C09088=1094.562,101.810,-61.706,176.099,17.273,152.460
C09089=1094.567,102.058,-61.724,176.101,17.273,152.459
C09090=1094.573,102.308,-61.742,176.104,17.274,152.459
C09091=1094.578,102.557,-61.761,176.106,17.275,152.459
C09092=1094.585,102.807,-61.779,176.108,17.276,152.458
C09093=1094.590,103.055,-61.798,176.111,17.277,152.458
C09094=1094.596,103.305,-61.816,176.113,17.277,152.458
C09095=1094.601,103.554,-61.835,176.116,17.279,152.457
C09096=1094.607,103.804,-61.853,176.119,17.279,152.457
C09097=1094.612,104.053,-61.871,176.121,17.280,152.457
C09098=1094.618,104.302,-61.890,176.123,17.281,152.457
C09099=1094.623,104.551,-61.909,176.126,17.281,152.456
C09100=1094.629,104.801,-61.926,176.128,17.283,152.456
C09101=1094.635,105.050,-61.946,176.131,17.284,152.456
C09102=1094.641,105.299,-61.963,176.133,17.284,152.455
C09103=1094.646,105.549,-61.983,176.136,17.285,152.455
C09104=1094.652,105.798,-62.000,176.138,17.286,152.455
C09105=1094.657,106.047,-62.019,176.141,17.287,152.454
C09106=1094.662,106.296,-62.037,176.144,17.288,152.454
C09107=1094.669,106.545,-62.056,176.145,17.288,152.454
C09108=1094.674,106.794,-62.075,176.148,17.289,152.453
C09109=1094.680,107.044,-62.093,176.151,17.290,152.453
C09110=1094.686,107.293,-62.112,176.153,17.291,152.453
C09111=1094.691,107.542,-62.130,176.156,17.292,152.452
C09112=1094.697,107.792,-62.149,176.158,17.292,152.452
C09113=1094.702,108.041,-62.168,176.161,17.293,152.452
C09114=1094.708,108.290,-62.186,176.164,17.294,152.451
C09115=1094.714,108.540,-62.205,176.166,17.295,152.451
C09116=1094.719,108.788,-62.223,176.169,17.296,152.451
C09117=1094.725,109.038,-62.243,176.171,17.296,152.450
C09118=1094.731,109.288,-62.261,176.173,17.297,152.450
C09119=1094.736,109.536,-62.279,176.176,17.298,152.450
C09120=1094.742,109.786,-62.299,176.178,17.299,152.449
C09121=1094.748,110.035,-62.317,176.181,17.300,152.449
C09122=1094.753,110.284,-62.335,176.184,17.301,152.449
C09123=1094.759,110.533,-62.355,176.186,17.301,152.449
C09124=1094.765,110.783,-62.373,176.189,17.302,152.448
C09125=1094.770,111.032,-62.391,176.191,17.302,152.448
C09126=1094.776,111.281,-62.411,176.194,17.303,152.447
C09127=1094.782,111.556,-62.431,176.197,17.304,152.447
C09128=1094.789,111.832,-62.452,176.199,17.305,152.447
C09129=1094.795,112.107,-62.473,176.202,17.306,152.446
C09130=1094.801,112.383,-62.494,176.205,17.307,152.446
C09131=1094.807,112.632,-62.512,176.207,17.307,152.446
C09132=1094.812,112.882,-62.531,176.210,17.308,152.445
C09133=1094.818,113.131,-62.550,176.213,17.309,152.445
C09134=1094.824,113.381,-62.570,176.215,17.310,152.445
C09135=1094.829,113.629,-62.588,176.218,17.311,152.444
C09136=1094.835,113.878,-62.607,176.220,17.311,152.444
C09137=1094.841,114.128,-62.626,176.223,17.312,152.443
C09138=1094.846,114.377,-62.645,176.226,17.313,152.443
C09139=1094.852,114.626,-62.664,176.228,17.313,152.443
C09140=1094.858,114.876,-62.682,176.231,17.314,152.443
C09141=1094.863,115.125,-62.701,176.234,17.315,152.442
C09142=1094.868,115.374,-62.720,176.236,17.316,152.442
C09143=1094.874,115.623,-62.740,176.239,17.316,152.441
C09144=1094.879,115.872,-62.759,176.241,17.318,152.441
C09145=1094.885,116.122,-62.778,176.243,17.318,152.441
C09146=1094.891,116.371,-62.797,176.246,17.319,152.441
C09147=1094.896,116.620,-62.816,176.249,17.320,152.440
C09148=1094.901,116.869,-62.835,176.251,17.321,152.440
C09149=1094.907,117.119,-62.854,176.254,17.321,152.439
C09150=1094.912,117.367,-62.873,176.257,17.322,152.439
C09151=1094.918,117.617,-62.893,176.259,17.323,152.439
C09152=1094.924,117.866,-62.912,176.262,17.323,152.438
C09153=1094.929,118.116,-62.931,176.265,17.325,152.438
C09154=1094.934,118.364,-62.950,176.267,17.325,152.438
C09155=1094.940,118.614,-62.969,176.270,17.326,152.437
C09156=1094.946,118.863,-62.988,176.273,17.327,152.437
C09157=1094.952,119.112,-63.007,176.275,17.327,152.437
C09158=1094.957,119.361,-63.026,176.278,17.328,152.436
C09159=1094.963,119.611,-63.045,176.280,17.328,152.436
C09160=1094.969,119.859,-63.065,176.283,17.329,152.436
C09161=1094.974,120.108,-63.084,176.286,17.330,152.435
C09162=1094.980,120.357,-63.103,176.287,17.331,152.435
C09163=1094.985,120.607,-63.122,176.290,17.331,152.434
C09164=1094.991,120.856,-63.142,176.293,17.332,152.434
C09165=1094.997,121.106,-63.161,176.295,17.333,152.434
C09166=1095.002,121.355,-63.180,176.298,17.333,152.433
C09167=1095.007,121.604,-63.200,176.301,17.334,152.433
C09168=1095.013,121.853,-63.220,176.303,17.335,152.433
C09169=1095.018,122.103,-63.239,176.306,17.336,152.432
C09170=1095.024,122.352,-63.258,176.309,17.336,152.432
C09171=1095.029,122.601,-63.277,176.311,17.337,152.432
C09172=1095.035,122.849,-63.297,176.314,17.338,152.431
C09173=1095.041,123.099,-63.316,176.317,17.338,152.431
C09174=1095.047,123.348,-63.335,176.319,17.339,152.430
C09175=1095.052,123.598,-63.355,176.322,17.339,152.430
C09176=1095.058,123.847,-63.375,176.325,17.340,152.430
C09177=1095.063,124.095,-63.394,176.327,17.341,152.429
C09178=1095.069,124.345,-63.413,176.330,17.342,152.429
C09179=1095.075,124.594,-63.432,176.333,17.342,152.429
C09180=1095.081,124.843,-63.452,176.336,17.343,152.428
C09181=1095.086,125.092,-63.471,176.338,17.343,152.428
C09182=1095.092,125.342,-63.490,176.341,17.345,152.427
C09183=1095.098,125.591,-63.510,176.344,17.345,152.427
C09184=1095.103,125.840,-63.530,176.346,17.345,152.427
C09185=1095.108,126.089,-63.549,176.349,17.346,152.426
C09186=1095.114,126.338,-63.569,176.352,17.347,152.426
C09187=1095.120,126.587,-63.588,176.354,17.347,152.425
C09188=1095.125,126.837,-63.608,176.357,17.348,152.425
C09189=1095.131,127.086,-63.628,176.360,17.349,152.425
C09190=1095.137,127.335,-63.647,176.362,17.349,152.424
C09191=1095.144,127.610,-63.669,176.365,17.350,152.424
C09192=1095.150,127.887,-63.691,176.368,17.350,152.423
C09193=1095.156,128.161,-63.712,176.371,17.351,152.423
C09194=1095.162,128.437,-63.733,176.374,17.352,152.422
C09195=1095.168,128.686,-63.753,176.377,17.353,152.422
C09196=1095.174,128.935,-63.772,176.380,17.353,152.422
C09197=1095.179,129.184,-63.793,176.383,17.354,152.421
C09198=1095.185,129.434,-63.812,176.386,17.354,152.421
C09199=1095.191,129.683,-63.832,176.389,17.355,152.420
C09200=1095.196,129.932,-63.851,176.391,17.355,152.420
C09201=1095.202,130.181,-63.871,176.394,17.356,152.420
C09202=1095.208,130.430,-63.891,176.397,17.357,152.419
C09203=1095.213,130.680,-63.911,176.399,17.357,152.419
C09204=1095.219,130.929,-63.930,176.402,17.358,152.418
C09205=1095.225,131.178,-63.950,176.405,17.358,152.418
C09206=1095.231,131.427,-63.970,176.407,17.359,152.418
C09207=1095.237,131.676,-63.990,176.410,17.359,152.417
C09208=1095.242,131.925,-64.010,176.413,17.360,152.417
C09209=1095.248,132.175,-64.029,176.416,17.361,152.416
C09210=1095.254,132.423,-64.049,176.418,17.361,152.416
C09211=1095.259,132.673,-64.070,176.421,17.362,152.415
C09212=1095.265,132.922,-64.089,176.424,17.363,152.415
C09213=1095.271,133.171,-64.109,176.426,17.363,152.415
C09214=1095.275,133.421,-64.129,176.429,17.364,152.414
C09215=1095.281,133.669,-64.149,176.432,17.364,152.414
C09216=1095.287,133.918,-64.169,176.434,17.364,152.413
C09217=1095.292,134.168,-64.189,176.437,17.365,152.413
C09218=1095.298,134.417,-64.209,176.440,17.366,152.413
C09219=1095.304,134.666,-64.229,176.443,17.367,152.412
C09220=1095.309,134.915,-64.248,176.446,17.367,152.412
C09221=1095.315,135.164,-64.268,176.449,17.367,152.411
C09222=1095.321,135.413,-64.289,176.452,17.368,152.411
C09223=1095.327,135.662,-64.309,176.454,17.368,152.410
C09224=1095.332,135.912,-64.329,176.457,17.369,152.410
C09225=1095.338,136.161,-64.349,176.460,17.370,152.410
C09226=1095.343,136.410,-64.369,176.463,17.370,152.409
C09227=1095.349,136.658,-64.389,176.465,17.371,152.409
C09228=1095.354,136.908,-64.409,176.468,17.371,152.408
C09229=1095.360,137.157,-64.429,176.471,17.372,152.408
C09230=1095.366,137.406,-64.449,176.473,17.372,152.408
C09231=1095.371,137.655,-64.470,176.476,17.373,152.407
C09232=1095.378,137.905,-64.490,176.479,17.373,152.407
C09233=1095.383,138.154,-64.510,176.482,17.374,152.406
C09234=1095.389,138.403,-64.530,176.485,17.374,152.406
C09235=1095.394,138.652,-64.550,176.488,17.375,152.405
C09236=1095.400,138.901,-64.570,176.491,17.376,152.405
C09237=1095.405,139.150,-64.591,176.494,17.376,152.404
C09238=1095.411,139.399,-64.611,176.496,17.376,152.404
C09239=1095.416,139.649,-64.631,176.499,17.377,152.404
C09240=1095.422,139.897,-64.651,176.502,17.378,152.403
C09241=1095.427,140.147,-64.671,176.504,17.378,152.403
C09242=1095.433,140.395,-64.691,176.507,17.378,152.402
C09243=1095.439,140.645,-64.712,176.510,17.379,152.402
C09244=1095.444,140.894,-64.733,176.513,17.380,152.401
C09245=1095.450,141.143,-64.752,176.516,17.380,152.401
C09246=1095.456,141.392,-64.773,176.519,17.381,152.401
C09247=1095.462,141.641,-64.793,176.522,17.382,152.400
C09248=1095.467,141.890,-64.814,176.525,17.382,152.400
C09249=1095.472,142.139,-64.834,176.527,17.382,152.399
C09250=1095.478,142.388,-64.854,176.530,17.383,152.399
C09251=1095.483,142.637,-64.875,176.533,17.384,152.398
C09252=1095.489,142.887,-64.896,176.536,17.384,152.398
C09253=1095.495,143.136,-64.915,176.538,17.384,152.397
C09254=1095.500,143.385,-64.936,176.541,17.385,152.397
C09255=1095.506,143.661,-64.959,176.545,17.385,152.396
C09256=1095.512,143.936,-64.981,176.548,17.386,152.396
C09257=1095.519,144.211,-65.004,176.551,17.386,152.395
C09258=1095.525,144.487,-65.026,176.554,17.387,152.395
C09259=1095.531,144.736,-65.047,176.557,17.388,152.395
C09260=1095.536,144.985,-65.067,176.560,17.388,152.394
C09261=1095.542,145.234,-65.088,176.562,17.388,152.394
C09262=1095.548,145.483,-65.108,176.565,17.389,152.393
C09263=1095.553,145.732,-65.129,176.569,17.389,152.393
C09264=1095.559,145.981,-65.149,176.572,17.390,152.392
C09265=1095.565,146.230,-65.170,176.574,17.390,152.392
C09266=1095.570,146.480,-65.191,176.577,17.391,152.391
C09267=1095.576,146.729,-65.211,176.580,17.391,152.391
C09268=1095.582,146.978,-65.231,176.583,17.392,152.390
C09269=1095.587,147.226,-65.253,176.585,17.392,152.390
C09270=1095.592,147.475,-65.273,176.588,17.393,152.390
C09271=1095.598,147.725,-65.294,176.592,17.393,152.389
C09272=1095.604,147.974,-65.314,176.595,17.394,152.389
C09273=1095.610,148.222,-65.335,176.597,17.393,152.388
C09274=1095.615,148.472,-65.356,176.600,17.394,152.388
C09275=1095.621,148.721,-65.377,176.603,17.395,152.387
C09276=1095.626,148.971,-65.397,176.606,17.395,152.387
C09277=1095.633,149.219,-65.418,176.608,17.395,152.386
C09278=1095.638,149.468,-65.439,176.612,17.396,152.386
C09279=1095.644,149.718,-65.460,176.615,17.397,152.385
C09280=1095.649,149.967,-65.480,176.618,17.397,152.385
C09281=1095.654,150.215,-65.501,176.621,17.398,152.384
C09282=1095.660,150.464,-65.522,176.623,17.398,152.384
C09283=1095.666,150.714,-65.543,176.626,17.398,152.383
C09284=1095.671,150.963,-65.564,176.629,17.399,152.383
C09285=1095.677,151.212,-65.584,176.632,17.400,152.382
C09286=1095.682,151.461,-65.605,176.635,17.399,152.382
C09287=1095.689,151.710,-65.626,176.638,17.400,152.382
C09288=1095.694,151.959,-65.647,176.641,17.400,152.381
C09289=1095.699,152.208,-65.668,176.644,17.401,152.381
C09290=1095.705,152.457,-65.689,176.647,17.402,152.380
C09291=1095.711,152.706,-65.710,176.649,17.402,152.380
C09292=1095.716,152.955,-65.731,176.653,17.402,152.379
C09293=1095.722,153.205,-65.752,176.656,17.403,152.379
C09294=1095.727,153.453,-65.773,176.659,17.403,152.378
C09295=1095.733,153.702,-65.794,176.661,17.403,152.378
C09296=1095.739,153.952,-65.815,176.664,17.404,152.377
C09297=1095.744,154.201,-65.836,176.667,17.404,152.377
C09298=1095.750,154.449,-65.857,176.671,17.405,152.376
C09299=1095.756,154.699,-65.878,176.674,17.405,152.376
C09300=1095.761,154.948,-65.899,176.676,17.405,152.375
C09301=1095.766,155.197,-65.920,176.679,17.405,152.375
C09302=1095.773,155.446,-65.941,176.682,17.406,152.374
C09303=1095.778,155.695,-65.962,176.686,17.407,152.374
C09304=1095.783,155.944,-65.983,176.688,17.407,152.373
C09305=1095.789,156.193,-66.004,176.691,17.407,152.373
C09306=1095.795,156.442,-66.025,176.694,17.408,152.372
C09307=1095.800,156.690,-66.047,176.697,17.408,152.372
C09308=1095.806,156.940,-66.068,176.700,17.409,152.371
C09309=1095.812,157.189,-66.089,176.703,17.409,152.371
C09310=1095.817,157.438,-66.109,176.706,17.409,152.370
C09311=1095.823,157.687,-66.131,176.709,17.410,152.370
C09312=1095.828,157.936,-66.153,176.712,17.410,152.369
C09313=1095.834,158.186,-66.174,176.715,17.411,152.369
C09314=1095.839,158.434,-66.195,176.718,17.411,152.368
C09315=1095.845,158.683,-66.216,176.721,17.411,152.368
C09316=1095.851,158.933,-66.237,176.724,17.412,152.367
C09317=1095.856,159.181,-66.259,176.727,17.412,152.367
C09318=1095.863,159.430,-66.280,176.730,17.412,152.366
C09319=1095.868,159.706,-66.304,176.734,17.413,152.366
C09320=1095.874,159.981,-66.327,176.737,17.413,152.365
C09321=1095.881,160.255,-66.350,176.740,17.413,152.364
C09322=1095.888,160.531,-66.374,176.743,17.414,152.364
C09323=1095.892,160.780,-66.396,176.746,17.414,152.363
C09324=1095.898,161.029,-66.417,176.750,17.415,152.363
C09325=1095.904,161.278,-66.438,176.752,17.414,152.362
C09326=1095.909,161.527,-66.459,176.755,17.415,152.362
C09327=1095.916,161.776,-66.481,176.758,17.415,152.361
C09328=1095.920,162.025,-66.503,176.761,17.416,152.361
C09329=1095.927,162.274,-66.525,176.764,17.417,152.360
C09330=1095.931,162.524,-66.546,176.768,17.417,152.360
C09331=1095.937,162.772,-66.567,176.770,17.417,152.359
C09332=1095.943,163.021,-66.589,176.773,17.417,152.359
C09333=1095.948,163.270,-66.610,176.776,17.418,152.358
C09334=1095.954,163.519,-66.632,176.779,17.419,152.358
C09335=1095.959,163.768,-66.654,176.783,17.419,152.357
C09336=1095.964,164.017,-66.675,176.786,17.419,152.357
C09337=1095.970,164.266,-66.696,176.788,17.419,152.356
C09338=1095.975,164.515,-66.718,176.791,17.420,152.356
C09339=1095.981,164.764,-66.740,176.795,17.420,152.355
C09340=1095.986,165.013,-66.762,176.798,17.421,152.355
C09341=1095.992,165.262,-66.783,176.801,17.421,152.354
C09342=1095.997,165.511,-66.805,176.804,17.421,152.354
C09343=1096.003,165.760,-66.827,176.806,17.422,152.353
C09344=1096.008,166.009,-66.848,176.809,17.422,152.353
C09345=1096.013,166.258,-66.870,176.813,17.422,152.352
C09346=1096.019,166.507,-66.891,176.816,17.423,152.352
C09347=1096.024,166.756,-66.913,176.819,17.423,152.351
C09348=1096.030,167.005,-66.935,176.822,17.424,152.351
C09349=1096.035,167.254,-66.957,176.825,17.423,152.350
C09350=1096.041,167.503,-66.978,176.828,17.424,152.350
C09351=1096.046,167.752,-67.000,176.831,17.425,152.349
C09352=1096.052,168.001,-67.022,176.834,17.425,152.349
C09353=1096.058,168.251,-67.044,176.837,17.425,152.348
C09354=1096.063,168.499,-67.065,176.841,17.425,152.348
C09355=1096.069,168.749,-67.088,176.843,17.425,152.347
C09356=1096.074,168.997,-67.109,176.846,17.426,152.347
C09357=1096.080,169.247,-67.131,176.849,17.426,152.346
C09358=1096.086,169.494,-67.153,176.853,17.427,152.345
C09359=1096.091,169.744,-67.175,176.856,17.427,152.345
C09360=1096.097,169.992,-67.197,176.859,17.427,152.344
C09361=1096.102,170.242,-67.219,176.862,17.428,152.344
C09362=1096.108,170.491,-67.240,176.865,17.428,152.343
C09363=1096.113,170.740,-67.262,176.868,17.428,152.343
C09364=1096.119,170.989,-67.284,176.871,17.428,152.342
C09365=1096.124,171.237,-67.307,176.874,17.429,152.342
C09366=1096.130,171.487,-67.329,176.878,17.429,152.341
C09367=1096.135,171.735,-67.350,176.881,17.429,152.341
C09368=1096.141,171.985,-67.372,176.884,17.430,152.340
C09369=1096.147,172.234,-67.395,176.887,17.430,152.340
C09370=1096.152,172.482,-67.417,176.890,17.430,152.339
C09371=1096.158,172.732,-67.438,176.893,17.430,152.338
C09372=1096.164,172.981,-67.460,176.896,17.431,152.338
C09373=1096.169,173.229,-67.483,176.900,17.431,152.337
C09374=1096.175,173.478,-67.505,176.903,17.432,152.337
C09375=1096.180,173.728,-67.527,176.906,17.432,152.336
C09376=1096.186,173.976,-67.549,176.908,17.432,152.336
C09377=1096.192,174.225,-67.571,176.911,17.432,152.335
C09378=1096.197,174.475,-67.593,176.915,17.432,152.335
C09379=1096.203,174.723,-67.615,176.918,17.433,152.334
C09380=1096.208,174.972,-67.637,176.921,17.433,152.334
C09381=1096.215,175.222,-67.659,176.924,17.433,152.333
C09382=1096.220,175.470,-67.682,176.928,17.434,152.332
C09383=1096.226,175.745,-67.707,176.931,17.434,152.332
C09384=1096.232,176.020,-67.731,176.935,17.434,152.331
C09385=1096.239,176.294,-67.755,176.938,17.434,152.330
C09386=1096.245,176.570,-67.780,176.941,17.434,152.330
C09387=1096.250,176.818,-67.802,176.945,17.434,152.329
C09388=1096.256,177.067,-67.824,176.948,17.435,152.329
C09389=1096.262,177.316,-67.846,176.951,17.435,152.328
C09390=1096.267,177.565,-67.869,176.954,17.435,152.328
C09391=1096.273,177.814,-67.891,176.958,17.436,152.327
C09392=1096.279,178.063,-67.914,176.961,17.436,152.327
C09393=1096.284,178.312,-67.936,176.964,17.435,152.326
C09394=1096.291,178.561,-67.958,176.967,17.436,152.325
C09395=1096.295,178.810,-67.980,176.970,17.436,152.325
C09396=1096.301,179.059,-68.003,176.973,17.436,152.324
C09397=1096.307,179.308,-68.025,176.977,17.437,152.324
C09398=1096.313,179.557,-68.048,176.980,17.437,152.323
C09399=1096.318,179.805,-68.069,176.983,17.437,152.322
C09400=1096.324,180.054,-68.092,176.987,17.437,152.322
C09401=1096.330,180.303,-68.115,176.989,17.437,152.321
C09402=1096.336,180.552,-68.137,176.992,17.437,152.321
C09403=1096.341,180.801,-68.160,176.996,17.438,152.320
C09404=1096.347,181.050,-68.183,176.999,17.438,152.320
C09405=1096.353,181.299,-68.204,177.002,17.438,152.319
C09406=1096.358,181.548,-68.227,177.006,17.438,152.318
C09407=1096.364,181.797,-68.250,177.009,17.439,152.318
C09408=1096.369,182.046,-68.272,177.012,17.439,152.317
C09409=1096.376,182.295,-68.295,177.015,17.439,152.317
C09410=1096.382,182.544,-68.318,177.018,17.439,152.316
C09411=1096.387,182.793,-68.340,177.021,17.439,152.315
C09412=1096.392,183.041,-68.362,177.025,17.439,152.315
C09413=1096.399,183.290,-68.385,177.028,17.440,152.314
C09414=1096.404,183.539,-68.408,177.031,17.439,152.314
C09415=1096.410,183.788,-68.430,177.035,17.440,152.313
C09416=1096.416,184.037,-68.453,177.038,17.440,152.312
C09417=1096.421,184.286,-68.476,177.041,17.440,152.312
C09418=1096.428,184.535,-68.498,177.045,17.440,152.311
C09419=1096.433,184.784,-68.520,177.048,17.441,152.311
C09420=1096.439,185.033,-68.543,177.051,17.440,152.310
C09421=1096.445,185.282,-68.566,177.054,17.440,152.309
C09422=1096.450,185.530,-68.589,177.057,17.441,152.309
C09423=1096.456,185.779,-68.612,177.060,17.441,152.308
C09424=1096.461,186.028,-68.635,177.064,17.441,152.308
C09425=1096.467,186.277,-68.657,177.067,17.442,152.307
C09426=1096.472,186.527,-68.680,177.070,17.442,152.307
C09427=1096.477,186.775,-68.703,177.074,17.442,152.306
C09428=1096.483,187.024,-68.726,177.077,17.442,152.305
C09429=1096.488,187.273,-68.749,177.080,17.443,152.305
C09430=1096.494,187.522,-68.772,177.083,17.443,152.304
C09431=1096.500,187.770,-68.795,177.087,17.443,152.304
C09432=1096.505,188.019,-68.818,177.090,17.444,152.303
C09433=1096.511,188.268,-68.841,177.093,17.444,152.302
C09434=1096.516,188.517,-68.864,177.096,17.443,152.302
C09435=1096.521,188.766,-68.886,177.099,17.444,152.301
C09436=1096.527,189.015,-68.909,177.102,17.444,152.301
C09437=1096.532,189.264,-68.932,177.106,17.444,152.300
C09438=1096.538,189.513,-68.955,177.109,17.444,152.300
C09439=1096.544,189.762,-68.978,177.112,17.445,152.299
C09440=1096.549,190.011,-69.001,177.116,17.445,152.298
C09441=1096.555,190.259,-69.025,177.119,17.445,152.298
C09442=1096.561,190.508,-69.048,177.122,17.445,152.297
C09443=1096.566,190.756,-69.071,177.126,17.445,152.297
C09444=1096.572,191.005,-69.094,177.129,17.446,152.296
C09445=1096.577,191.255,-69.117,177.132,17.446,152.295
C09446=1096.582,191.503,-69.140,177.136,17.446,152.295
C09447=1096.589,191.778,-69.166,177.139,17.446,152.294
C09448=1096.595,192.052,-69.191,177.142,17.446,152.293
C09449=1096.601,192.327,-69.217,177.146,17.446,152.293
C09450=1096.607,192.601,-69.242,177.150,17.447,152.292
C09451=1096.613,192.850,-69.265,177.154,17.447,152.291
C09452=1096.619,193.099,-69.288,177.157,17.447,152.291
C09453=1096.624,193.348,-69.312,177.160,17.447,152.290
C09454=1096.630,193.597,-69.335,177.164,17.448,152.290
C09455=1096.635,193.846,-69.358,177.166,17.447,152.289
C09456=1096.641,194.094,-69.381,177.170,17.447,152.288
C09457=1096.646,194.344,-69.405,177.173,17.448,152.288
C09458=1096.652,194.593,-69.428,177.176,17.448,152.287
C09459=1096.658,194.841,-69.451,177.180,17.448,152.287
C09460=1096.664,195.090,-69.475,177.183,17.448,152.286
C09461=1096.669,195.339,-69.498,177.186,17.448,152.285
C09462=1096.675,195.588,-69.521,177.190,17.448,152.285
C09463=1096.680,195.837,-69.544,177.193,17.449,152.284
C09464=1096.686,196.085,-69.568,177.196,17.449,152.284
C09465=1096.691,196.334,-69.591,177.200,17.449,152.283
C09466=1096.697,196.583,-69.614,177.203,17.449,152.282
C09467=1096.702,196.832,-69.638,177.206,17.449,152.282
C09468=1096.708,197.081,-69.661,177.210,17.449,152.281
C09469=1096.714,197.329,-69.684,177.213,17.450,152.280
C09470=1096.719,197.578,-69.708,177.216,17.450,152.280
C09471=1096.725,197.828,-69.732,177.220,17.450,152.279
C09472=1096.731,198.076,-69.755,177.223,17.450,152.279
C09473=1096.736,198.325,-69.779,177.227,17.450,152.278
C09474=1096.742,198.574,-69.802,177.230,17.450,152.277
C09475=1096.748,198.822,-69.826,177.233,17.450,152.277
C09476=1096.753,199.072,-69.849,177.237,17.451,152.276
C09477=1096.759,199.320,-69.873,177.240,17.451,152.275
C09478=1096.765,199.569,-69.896,177.243,17.451,152.275
C09479=1096.771,199.818,-69.920,177.247,17.451,152.274
C09480=1096.777,200.067,-69.943,177.250,17.451,152.274
C09481=1096.783,200.315,-69.967,177.254,17.451,152.273
C09482=1096.788,200.564,-69.991,177.257,17.451,152.272
C09483=1096.794,200.813,-70.014,177.261,17.451,152.272
C09484=1096.799,201.062,-70.038,177.264,17.451,152.271
C09485=1096.805,201.311,-70.062,177.267,17.452,152.270
C09486=1096.811,201.560,-70.085,177.271,17.452,152.270
C09487=1096.816,201.808,-70.109,177.274,17.452,152.269
C09488=1096.822,202.057,-70.133,177.277,17.451,152.269
C09489=1096.827,202.306,-70.156,177.280,17.451,152.268
C09490=1096.834,202.555,-70.180,177.284,17.452,152.267
C09491=1096.839,202.804,-70.204,177.287,17.451,152.267
C09492=1096.845,203.052,-70.227,177.290,17.452,152.266
C09493=1096.850,203.301,-70.252,177.294,17.452,152.265
C09494=1096.856,203.550,-70.275,177.297,17.452,152.265
C09495=1096.861,203.798,-70.299,177.301,17.452,152.264
C09496=1096.867,204.048,-70.323,177.304,17.452,152.263
C09497=1096.873,204.297,-70.346,177.307,17.452,152.263
C09498=1096.878,204.545,-70.371,177.311,17.453,152.262
C09499=1096.884,204.793,-70.394,177.314,17.453,152.262
C09500=1096.889,205.043,-70.418,177.318,17.454,152.261
C09501=1096.895,205.292,-70.442,177.322,17.453,152.260
C09502=1096.901,205.540,-70.466,177.325,17.453,152.260
C09503=1096.906,205.789,-70.490,177.328,17.454,152.259
C09504=1096.912,206.038,-70.514,177.332,17.454,152.258
C09505=1096.918,206.286,-70.538,177.335,17.454,152.258
C09506=1096.923,206.535,-70.562,177.339,17.454,152.257
C09507=1096.929,206.784,-70.586,177.342,17.454,152.257
C09508=1096.935,207.033,-70.609,177.346,17.454,152.256
C09509=1096.940,207.282,-70.634,177.349,17.454,152.255
C09510=1096.946,207.531,-70.658,177.352,17.454,152.255
C09511=1096.969,208.543,-70.756,177.400,17.473,152.249
C09512=1096.977,208.915,-70.792,177.405,17.474,152.249
C09513=1096.986,209.287,-70.828,177.410,17.476,152.248
C09514=1096.994,209.658,-70.865,177.415,17.477,152.247
C09515=1097.002,210.030,-70.901,177.420,17.479,152.247
C09516=1097.008,210.280,-70.926,177.423,17.479,152.246
C09517=1097.013,210.528,-70.950,177.426,17.480,152.246
C09518=1097.019,210.777,-70.975,177.430,17.482,152.246
C09519=1097.025,211.026,-70.999,177.433,17.482,152.245
C09520=1097.030,211.275,-71.023,177.436,17.483,152.245
C09521=1097.036,211.524,-71.048,177.439,17.485,152.244
C09522=1097.041,211.772,-71.073,177.442,17.486,152.244
C09523=1097.047,212.020,-71.097,177.445,17.486,152.244
C09524=1097.053,212.270,-71.122,177.449,17.488,152.243
C09525=1097.058,212.518,-71.146,177.452,17.489,152.243
C09526=1097.065,212.767,-71.170,177.455,17.489,152.242
C09527=1097.070,213.015,-71.195,177.459,17.491,152.242
C09528=1097.076,213.265,-71.220,177.462,17.491,152.241
C09529=1097.081,213.513,-71.244,177.465,17.492,152.241
C09530=1097.086,213.762,-71.269,177.469,17.494,152.241
C09531=1097.092,214.011,-71.294,177.472,17.494,152.240
C09532=1097.097,214.259,-71.319,177.475,17.495,152.240
C09533=1097.103,214.509,-71.343,177.478,17.497,152.239
C09534=1097.109,214.757,-71.368,177.481,17.497,152.239
C09535=1097.114,215.005,-71.392,177.484,17.498,152.239
C09536=1097.120,215.254,-71.417,177.488,17.500,152.238
C09537=1097.126,215.502,-71.442,177.491,17.501,152.238
C09538=1097.132,215.752,-71.467,177.494,17.501,152.237
C09539=1097.136,216.001,-71.491,177.498,17.503,152.237
C09540=1097.142,216.249,-71.517,177.501,17.504,152.237
C09541=1097.148,216.498,-71.541,177.504,17.505,152.236
C09542=1097.154,216.747,-71.566,177.507,17.506,152.236
C09543=1097.159,216.995,-71.591,177.510,17.507,152.235
C09544=1097.165,217.244,-71.615,177.514,17.508,152.235
C09545=1097.171,217.492,-71.640,177.517,17.509,152.235
C09546=1097.176,217.742,-71.665,177.520,17.510,152.234
C09547=1097.182,217.990,-71.690,177.524,17.511,152.234
C09548=1097.187,218.239,-71.715,177.527,17.512,152.233
C09549=1097.193,218.487,-71.740,177.530,17.513,152.233
C09550=1097.199,218.737,-71.765,177.534,17.514,152.232
C09551=1097.204,218.985,-71.790,177.537,17.515,152.232
C09552=1097.210,219.234,-71.815,177.541,17.516,152.232
C09553=1097.215,219.482,-71.840,177.544,17.517,152.231
C09554=1097.221,219.731,-71.864,177.546,17.518,152.231
C09555=1097.227,219.980,-71.890,177.550,17.519,152.230
C09556=1097.232,220.229,-71.915,177.553,17.520,152.230
C09557=1097.238,220.478,-71.940,177.556,17.521,152.230
C09558=1097.244,220.726,-71.965,177.560,17.522,152.229
C09559=1097.250,220.975,-71.990,177.563,17.523,152.229
C09560=1097.255,221.223,-72.015,177.567,17.525,152.228
C09561=1097.260,221.472,-72.040,177.570,17.525,152.228
C09562=1097.267,221.721,-72.065,177.573,17.526,152.228
C09563=1097.272,221.969,-72.090,177.577,17.527,152.227
C09564=1097.281,222.345,-72.128,177.581,17.529,152.227
C09565=1097.288,222.721,-72.167,177.586,17.531,152.226
C09566=1097.297,223.097,-72.205,177.591,17.532,152.225
C09567=1097.305,223.473,-72.243,177.596,17.534,152.225
C09568=1097.312,223.721,-72.268,177.600,17.535,152.224
C09569=1097.317,223.971,-72.293,177.603,17.536,152.224
C09570=1097.322,224.219,-72.318,177.606,17.537,152.224
C09571=1097.329,224.467,-72.344,177.609,17.538,152.223
C09572=1097.333,224.716,-72.369,177.612,17.539,152.223
C09573=1097.339,224.965,-72.394,177.616,17.540,152.222
C09574=1097.345,225.214,-72.420,177.619,17.541,152.222
C09575=1097.350,225.462,-72.445,177.622,17.542,152.222
C09576=1097.356,225.711,-72.471,177.626,17.544,152.221
C09577=1097.362,225.960,-72.496,177.629,17.544,152.221
C09578=1097.367,226.208,-72.521,177.633,17.546,152.220
C09579=1097.373,226.457,-72.547,177.636,17.547,152.220
C09580=1097.379,226.706,-72.573,177.639,17.548,152.220
C09581=1097.384,226.954,-72.597,177.642,17.549,152.219
C09582=1097.389,227.203,-72.623,177.645,17.550,152.219
C09583=1097.396,227.452,-72.648,177.649,17.551,152.218
C09584=1097.401,227.701,-72.674,177.652,17.552,152.218
C09585=1097.407,227.949,-72.699,177.656,17.554,152.218
C09586=1097.412,228.198,-72.725,177.659,17.554,152.217
C09587=1097.418,228.446,-72.750,177.662,17.555,152.217
C09588=1097.423,228.695,-72.776,177.665,17.557,152.216
C09589=1097.429,228.943,-72.801,177.668,17.558,152.216
C09590=1097.435,229.192,-72.827,177.672,17.559,152.216
C09591=1097.441,229.441,-72.853,177.675,17.560,152.215
C09592=1097.446,229.689,-72.878,177.679,17.561,152.215
C09593=1097.452,229.938,-72.904,177.682,17.562,152.214
C09594=1097.458,230.187,-72.929,177.685,17.563,152.214
C09595=1097.463,230.435,-72.956,177.689,17.564,152.214
C09596=1097.470,230.684,-72.981,177.692,17.565,152.213
C09597=1097.475,230.932,-73.007,177.695,17.567,152.213
C09598=1097.480,231.181,-73.033,177.698,17.568,152.213
C09599=1097.486,231.430,-73.058,177.702,17.569,152.212
C09600=1097.492,231.679,-73.084,177.705,17.570,152.212
C09601=1097.497,231.927,-73.110,177.709,17.571,152.211
C09602=1097.503,232.176,-73.135,177.712,17.572,152.211
C09603=1097.509,232.424,-73.162,177.715,17.574,152.211
C09604=1097.514,232.673,-73.188,177.718,17.574,152.210
C09605=1097.519,232.922,-73.214,177.721,17.575,152.210
C09606=1097.525,233.170,-73.239,177.725,17.577,152.209
C09607=1097.531,233.418,-73.265,177.728,17.578,152.209
C09608=1097.536,233.667,-73.291,177.732,17.579,152.209
C09609=1097.542,233.916,-73.317,177.735,17.580,152.208
C09610=1097.548,234.165,-73.342,177.739,17.581,152.208
C09611=1097.553,234.413,-73.369,177.742,17.582,152.207
C09612=1097.559,234.662,-73.395,177.745,17.584,152.207
C09613=1097.564,234.911,-73.421,177.748,17.585,152.207
C09614=1097.570,235.159,-73.447,177.752,17.586,152.206
C09615=1097.576,235.408,-73.473,177.755,17.587,152.206
C09616=1097.584,235.775,-73.511,177.760,17.589,152.205
C09617=1097.592,236.143,-73.550,177.764,17.590,152.205
C09618=1097.600,236.509,-73.588,177.770,17.593,152.204
C09619=1097.608,236.878,-73.627,177.775,17.594,152.204
C09620=1097.615,237.126,-73.653,177.778,17.596,152.203
C09621=1097.620,237.374,-73.678,177.781,17.597,152.203
C09622=1097.625,237.622,-73.705,177.784,17.598,152.203
C09623=1097.631,237.871,-73.731,177.788,17.599,152.202
C09624=1097.637,238.120,-73.758,177.791,17.600,152.202
C09625=1097.642,238.369,-73.784,177.795,17.602,152.201
C09626=1097.648,238.617,-73.810,177.798,17.602,152.201
C09627=1097.653,238.866,-73.836,177.801,17.604,152.201
C09628=1097.659,239.114,-73.863,177.804,17.605,152.200
C09629=1097.665,239.363,-73.889,177.808,17.606,152.200
C09630=1097.670,239.612,-73.915,177.811,17.607,152.200
C09631=1097.677,239.860,-73.941,177.815,17.608,152.199
C09632=1097.682,240.109,-73.967,177.818,17.609,152.199
C09633=1097.688,240.357,-73.994,177.821,17.611,152.199
C09634=1097.693,240.605,-74.020,177.824,17.612,152.198
C09635=1097.699,240.854,-74.046,177.828,17.614,152.198
C09636=1097.704,241.103,-74.072,177.831,17.614,152.197
C09637=1097.710,241.351,-74.099,177.835,17.616,152.197
C09638=1097.716,241.599,-74.126,177.838,17.617,152.197
C09639=1097.721,241.848,-74.151,177.841,17.618,152.196
C09640=1097.727,242.097,-74.178,177.844,17.619,152.196
C09641=1097.733,242.345,-74.205,177.848,17.620,152.195
C09642=1097.739,242.593,-74.231,177.851,17.621,152.195
C09643=1097.743,242.843,-74.258,177.855,17.623,152.195
C09644=1097.749,243.091,-74.285,177.858,17.624,152.194
C09645=1097.755,243.339,-74.311,177.861,17.626,152.194
C09646=1097.761,243.588,-74.338,177.864,17.626,152.194
C09647=1097.766,243.837,-74.364,177.868,17.628,152.193
C09648=1097.772,244.085,-74.390,177.871,17.629,152.193
C09649=1097.778,244.333,-74.417,177.875,17.630,152.192
C09650=1097.783,244.582,-74.444,177.877,17.632,152.192
C09651=1097.788,244.830,-74.471,177.881,17.633,152.192
C09652=1097.794,245.079,-74.497,177.885,17.634,152.191
C09653=1097.800,245.328,-74.524,177.888,17.635,152.191
C09654=1097.805,245.576,-74.550,177.892,17.637,152.191
C09655=1097.811,245.825,-74.577,177.895,17.638,152.190
C09656=1097.817,246.074,-74.604,177.898,17.640,152.190
C09657=1097.823,246.322,-74.631,177.901,17.640,152.190
C09658=1097.828,246.571,-74.658,177.905,17.642,152.189
C09659=1097.834,246.819,-74.684,177.908,17.643,152.189
C09660=1097.839,247.068,-74.712,177.912,17.644,152.188
C09661=1097.845,247.317,-74.738,177.914,17.645,152.188
C09662=1097.851,247.565,-74.764,177.918,17.647,152.188
C09663=1097.856,247.814,-74.792,177.922,17.648,152.187
C09664=1097.861,248.062,-74.818,177.925,17.649,152.187
C09665=1097.867,248.310,-74.845,177.928,17.651,152.187
C09666=1097.872,248.559,-74.872,177.931,17.652,152.186
C09667=1097.878,248.807,-74.899,177.935,17.653,152.186
C09668=1097.886,249.168,-74.938,177.939,17.656,152.186
C09669=1097.895,249.528,-74.977,177.944,17.657,152.185
C09670=1097.902,249.889,-75.016,177.949,17.659,152.185
C09671=1097.910,250.249,-75.056,177.955,17.661,152.184
C09672=1097.916,250.497,-75.083,177.957,17.662,152.184
C09673=1097.921,250.746,-75.110,177.961,17.664,152.183
C09674=1097.927,250.994,-75.137,177.964,17.665,152.183
C09675=1097.932,251.243,-75.163,177.968,17.666,152.183
C09676=1097.937,251.491,-75.191,177.970,17.668,152.182
C09677=1097.944,251.740,-75.218,177.974,17.669,152.182
C09678=1097.949,251.988,-75.246,177.978,17.671,152.182
C09679=1097.955,252.237,-75.272,177.981,17.672,152.181
C09680=1097.960,252.485,-75.299,177.984,17.673,152.181
C09681=1097.966,252.734,-75.326,177.987,17.674,152.181
C09682=1097.971,252.982,-75.354,177.991,17.676,152.180
C09683=1097.977,253.231,-75.381,177.994,17.678,152.180
C09684=1097.983,253.480,-75.408,177.997,17.679,152.180
C09685=1097.989,253.727,-75.436,178.001,17.680,152.179
C09686=1097.994,253.976,-75.463,178.004,17.681,152.179
C09687=1097.999,254.224,-75.490,178.008,17.683,152.179
C09688=1098.005,254.473,-75.518,178.011,17.684,152.178
C09689=1098.011,254.721,-75.545,178.014,17.685,152.178
C09690=1098.016,254.970,-75.572,178.018,17.687,152.178
C09691=1098.022,255.218,-75.599,178.021,17.688,152.177
C09692=1098.027,255.467,-75.626,178.025,17.689,152.177
C09693=1098.034,255.716,-75.653,178.028,17.691,152.177
C09694=1098.039,255.964,-75.681,178.031,17.692,152.176
C09695=1098.044,256.212,-75.709,178.035,17.694,152.176
C09696=1098.050,256.460,-75.736,178.038,17.694,152.176
C09697=1098.056,256.709,-75.764,178.041,17.696,152.175
C09698=1098.062,256.957,-75.791,178.045,17.698,152.175
C09699=1098.067,257.206,-75.818,178.048,17.699,152.175
C09700=1098.074,257.454,-75.846,178.052,17.700,152.174
C09701=1098.079,257.703,-75.873,178.054,17.702,152.174
C09702=1098.084,257.951,-75.901,178.058,17.703,152.174
C09703=1098.090,258.199,-75.928,178.062,17.704,152.173
C09704=1098.096,258.448,-75.956,178.064,17.706,152.173
C09705=1098.101,258.696,-75.983,178.068,17.707,152.173
C09706=1098.107,258.945,-76.011,178.072,17.709,152.172
C09707=1098.113,259.193,-76.039,178.075,17.710,152.172
C09708=1098.118,259.442,-76.066,178.078,17.711,152.172
C09709=1098.124,259.690,-76.094,178.081,17.712,152.171
C09710=1098.129,259.939,-76.121,178.085,17.714,152.171
C09711=1098.136,260.187,-76.149,178.089,17.716,152.171
C09712=1098.141,260.436,-76.177,178.092,17.717,152.170
C09713=1098.147,260.684,-76.204,178.095,17.718,152.170
C09714=1098.153,260.932,-76.231,178.099,17.720,152.169
C09715=1098.159,261.181,-76.260,178.102,17.721,152.169
C09716=1098.164,261.429,-76.287,178.106,17.722,152.169
C09717=1098.170,261.677,-76.314,178.108,17.723,152.168
C09718=1098.176,261.926,-76.343,178.112,17.725,152.168
C09719=1098.181,262.174,-76.371,178.116,17.727,152.168
C09720=1098.190,262.531,-76.410,178.121,17.728,152.167
C09721=1098.197,262.889,-76.450,178.125,17.730,152.167
C09722=1098.207,263.247,-76.490,178.130,17.732,152.166
C09723=1098.215,263.605,-76.531,178.135,17.735,152.166
C09724=1098.220,263.853,-76.559,178.138,17.735,152.165
C09725=1098.227,264.101,-76.586,178.142,17.737,152.165
C09726=1098.232,264.349,-76.614,178.145,17.739,152.165
C09727=1098.238,264.598,-76.643,178.148,17.740,152.165
C09728=1098.243,264.847,-76.670,178.152,17.742,152.164
C09729=1098.248,265.095,-76.698,178.156,17.743,152.164
C09730=1098.254,265.343,-76.726,178.158,17.744,152.164
C09731=1098.259,265.591,-76.754,178.162,17.746,152.163
C09732=1098.265,265.840,-76.782,178.166,17.748,152.163
C09733=1098.271,266.088,-76.810,178.169,17.749,152.163
C09734=1098.276,266.336,-76.838,178.172,17.751,152.162
C09735=1098.282,266.585,-76.867,178.176,17.752,152.162
C09736=1098.287,266.833,-76.895,178.178,17.753,152.162
C09737=1098.293,267.082,-76.923,178.182,17.755,152.161
C09738=1098.299,267.330,-76.951,178.186,17.757,152.161
C09739=1098.305,267.579,-76.979,178.189,17.758,152.161
C09740=1098.310,267.827,-77.007,178.192,17.760,152.161
C09741=1098.316,268.075,-77.035,178.196,17.761,152.160
C09742=1098.321,268.323,-77.063,178.200,17.763,152.160
C09743=1098.328,268.572,-77.092,178.202,17.764,152.160
C09744=1098.333,268.820,-77.120,178.206,17.765,152.159
C09745=1098.339,269.068,-77.149,178.209,17.767,152.159
C09746=1098.344,269.316,-77.177,178.212,17.768,152.159
C09747=1098.350,269.565,-77.205,178.216,17.770,152.158
C09748=1098.355,269.813,-77.233,178.220,17.772,152.158
C09749=1098.361,270.062,-77.261,178.222,17.773,152.158
C09750=1098.367,270.309,-77.290,178.226,17.774,152.157
C09751=1098.373,270.558,-77.318,178.230,17.776,152.157
C09752=1098.378,270.806,-77.346,178.232,17.778,152.157
C09753=1098.384,271.055,-77.375,178.236,17.779,152.157
C09754=1098.390,271.302,-77.403,178.239,17.781,152.156
C09755=1098.395,271.551,-77.432,178.243,17.782,152.156
C09756=1098.400,271.800,-77.460,178.246,17.784,152.156
C09757=1098.406,272.048,-77.488,178.250,17.785,152.155
C09758=1098.413,272.296,-77.518,178.253,17.787,152.155
C09759=1098.418,272.544,-77.545,178.256,17.788,152.155
C09760=1098.424,272.793,-77.574,178.260,17.790,152.155
C09761=1098.429,273.041,-77.603,178.263,17.792,152.154
C09762=1098.435,273.290,-77.631,178.267,17.793,152.154
C09763=1098.440,273.538,-77.659,178.269,17.795,152.154
C09764=1098.446,273.786,-77.688,178.273,17.796,152.153
C09765=1098.452,274.035,-77.717,178.277,17.798,152.153
C09766=1098.457,274.282,-77.746,178.280,17.800,152.153
C09767=1098.463,274.531,-77.774,178.283,17.801,152.153
C09768=1098.468,274.779,-77.802,178.287,17.803,152.152
C09769=1098.475,275.027,-77.831,178.290,17.805,152.152
C09770=1098.480,275.276,-77.860,178.293,17.806,152.152
C09771=1098.486,275.524,-77.889,178.297,17.808,152.152
C09772=1098.494,275.885,-77.931,178.302,17.810,152.151
C09773=1098.502,276.245,-77.972,178.306,17.812,152.151
C09774=1098.510,276.605,-78.014,178.311,17.814,152.150
C09775=1098.519,276.965,-78.056,178.316,17.817,152.150
C09776=1098.524,277.213,-78.085,178.320,17.819,152.150
C09777=1098.529,277.462,-78.113,178.322,17.820,152.150
C09778=1098.536,277.710,-78.142,178.326,17.822,152.149
C09779=1098.540,277.958,-78.171,178.330,17.824,152.149
C09780=1098.547,278.206,-78.200,178.333,17.826,152.149
C09781=1098.553,278.455,-78.229,178.336,17.826,152.148
C09782=1098.557,278.703,-78.258,178.340,17.828,152.148
C09783=1098.564,278.951,-78.287,178.343,17.830,152.148
C09784=1098.569,279.200,-78.316,178.347,17.832,152.148
C09785=1098.575,279.448,-78.344,178.350,17.833,152.147
C09786=1098.580,279.696,-78.374,178.353,17.835,152.147
C09787=1098.586,279.944,-78.403,178.356,17.837,152.147
C09788=1098.593,280.192,-78.432,178.360,17.838,152.146
C09789=1098.597,280.441,-78.460,178.364,17.840,152.146
C09790=1098.603,280.689,-78.490,178.366,17.842,152.146
C09791=1098.609,280.937,-78.519,178.370,17.844,152.146
C09792=1098.615,281.185,-78.548,178.374,17.845,152.145
C09793=1098.620,281.433,-78.577,178.377,17.847,152.145
C09794=1098.626,281.682,-78.606,178.380,17.848,152.145
C09795=1098.632,281.930,-78.635,178.383,17.850,152.145
C09796=1098.636,282.178,-78.665,178.387,17.852,152.145
C09797=1098.643,282.426,-78.694,178.390,17.854,152.144
C09798=1098.648,282.675,-78.723,178.394,17.856,152.144
C09799=1098.654,282.923,-78.752,178.397,17.857,152.144
C09800=1098.659,283.170,-78.782,178.400,17.859,152.144
C09801=1098.665,283.419,-78.811,178.404,17.861,152.143
C09802=1098.671,283.668,-78.840,178.407,17.863,152.143
C09803=1098.676,283.916,-78.869,178.411,17.865,152.143
C09804=1098.681,284.164,-78.899,178.413,17.866,152.143
C09805=1098.687,284.412,-78.928,178.417,17.868,152.142
C09806=1098.693,284.660,-78.957,178.420,17.869,152.142
C09807=1098.699,284.909,-78.987,178.424,17.871,152.142
C09808=1098.705,285.157,-79.016,178.427,17.873,152.142
C09809=1098.710,285.405,-79.045,178.430,17.875,152.141
C09810=1098.715,285.653,-79.075,178.434,17.877,152.141
C09811=1098.722,285.901,-79.105,178.437,17.878,152.141
C09812=1098.727,286.149,-79.134,178.440,17.880,152.141
C09813=1098.733,286.398,-79.164,178.444,17.882,152.141
C09814=1098.738,286.645,-79.193,178.447,17.884,152.140
C09815=1098.744,286.893,-79.222,178.450,17.886,152.140
C09816=1098.749,287.142,-79.252,178.454,17.887,152.140
C09817=1098.756,287.390,-79.281,178.457,17.889,152.140
C09818=1098.761,287.638,-79.310,178.461,17.891,152.139
C09819=1098.767,287.886,-79.341,178.464,17.893,152.139
C09820=1098.773,288.135,-79.370,178.467,17.894,152.139
C09821=1098.778,288.382,-79.399,178.470,17.896,152.139
C09822=1098.784,288.631,-79.429,178.474,17.898,152.138
C09823=1098.789,288.879,-79.458,178.477,17.900,152.138
C09824=1098.799,289.248,-79.503,178.483,17.903,152.138
C09825=1098.807,289.618,-79.547,178.487,17.905,152.138
C09826=1098.815,289.988,-79.591,178.492,17.908,152.137
C09827=1098.824,290.357,-79.636,178.497,17.911,152.137
C09828=1098.829,290.606,-79.666,178.501,17.913,152.137
C09829=1098.835,290.854,-79.695,178.504,17.915,152.136
C09830=1098.840,291.102,-79.726,178.507,17.916,152.136
C09831=1098.846,291.350,-79.754,178.511,17.918,152.136
C09832=1098.852,291.598,-79.784,178.514,17.920,152.136
C09833=1098.857,291.846,-79.814,178.517,17.922,152.136
C09834=1098.863,292.094,-79.844,178.521,17.924,152.135
C09835=1098.869,292.342,-79.874,178.524,17.926,152.135
C09836=1098.874,292.591,-79.904,178.528,17.928,152.135
C09837=1098.880,292.839,-79.934,178.530,17.929,152.135
C09838=1098.886,293.087,-79.964,178.534,17.931,152.135
C09839=1098.891,293.335,-79.994,178.537,17.933,152.135
C09840=1098.897,293.583,-80.024,178.541,17.935,152.134
C09841=1098.902,293.831,-80.054,178.544,17.937,152.134
C09842=1098.908,294.079,-80.084,178.548,17.939,152.134
C09843=1098.914,294.328,-80.114,178.551,17.941,152.134
C09844=1098.920,294.576,-80.144,178.555,17.943,152.133
C09845=1098.925,294.823,-80.174,178.557,17.945,152.133
C09846=1098.931,295.072,-80.204,178.561,17.947,152.133
C09847=1098.937,295.320,-80.234,178.564,17.949,152.133
C09848=1098.942,295.568,-80.264,178.567,17.951,152.133
C09849=1098.948,295.816,-80.294,178.571,17.952,152.133
C09850=1098.954,296.064,-80.325,178.574,17.954,152.132
C09851=1098.959,296.312,-80.354,178.578,17.957,152.132
C09852=1098.965,296.560,-80.385,178.581,17.959,152.132
C09853=1098.971,296.808,-80.415,178.585,17.961,152.132
C09854=1098.977,297.056,-80.445,178.588,17.963,152.132
C09855=1098.982,297.304,-80.475,178.590,17.964,152.132
C09856=1098.987,297.552,-80.506,178.594,17.966,152.131
C09857=1098.993,297.801,-80.535,178.597,17.968,152.131
C09858=1098.999,298.048,-80.566,178.601,17.970,152.131
C09859=1099.005,298.296,-80.596,178.604,17.972,152.131
C09860=1099.010,298.544,-80.626,178.608,17.974,152.131
C09861=1099.015,298.792,-80.657,178.611,17.976,152.130
C09862=1099.021,299.041,-80.687,178.614,17.979,152.130
C09863=1099.027,299.289,-80.717,178.618,17.981,152.130
C09864=1099.032,299.537,-80.748,178.621,17.983,152.130
C09865=1099.038,299.784,-80.779,178.624,17.985,152.130
C09866=1099.044,300.032,-80.809,178.628,17.987,152.130
C09867=1099.049,300.280,-80.840,178.631,17.989,152.130
C09868=1099.054,300.529,-80.870,178.635,17.991,152.129
C09869=1099.060,300.777,-80.900,178.637,17.993,152.129
C09870=1099.065,301.025,-80.931,178.640,17.995,152.129
C09871=1099.071,301.273,-80.962,178.644,17.997,152.129
C09872=1099.077,301.521,-80.992,178.647,17.999,152.129
C09873=1099.082,301.769,-81.023,178.650,18.002,152.129
C09874=1099.088,302.017,-81.053,178.654,18.004,152.129
C09875=1099.094,302.265,-81.084,178.657,18.006,152.129
C09876=1099.102,302.648,-81.131,178.662,18.009,152.128
C09877=1099.111,303.032,-81.179,178.667,18.012,152.128
C09878=1099.119,303.415,-81.226,178.673,18.016,152.128
C09879=1099.128,303.799,-81.274,178.678,18.019,152.128
C09880=1099.134,304.047,-81.304,178.681,18.021,152.128
C09881=1099.139,304.295,-81.335,178.685,18.024,152.127
C09882=1099.146,304.543,-81.366,178.688,18.026,152.127
C09883=1099.151,304.791,-81.397,178.691,18.028,152.127
C09884=1099.156,305.039,-81.427,178.695,18.030,152.127
C09885=1099.162,305.287,-81.459,178.698,18.032,152.127
C09886=1099.168,305.535,-81.489,178.701,18.034,152.127
C09887=1099.173,305.783,-81.520,178.705,18.037,152.127
C09888=1099.179,306.031,-81.551,178.708,18.039,152.126
C09889=1099.184,306.279,-81.582,178.711,18.041,152.126
C09890=1099.190,306.527,-81.613,178.715,18.043,152.126
C09891=1099.195,306.775,-81.644,178.718,18.045,152.126
C09892=1099.201,307.023,-81.674,178.721,18.048,152.126
C09893=1099.208,307.271,-81.705,178.725,18.049,152.126
C09894=1099.213,307.519,-81.736,178.728,18.052,152.126
C09895=1099.218,307.767,-81.767,178.731,18.054,152.126
C09896=1099.224,308.015,-81.798,178.734,18.056,152.126
C09897=1099.230,308.263,-81.830,178.738,18.059,152.126
C09898=1099.236,308.511,-81.860,178.741,18.060,152.125
C09899=1099.241,308.759,-81.891,178.744,18.063,152.125
C09900=1099.248,309.007,-81.922,178.748,18.065,152.125
C09901=1099.253,309.255,-81.953,178.751,18.067,152.125
C09902=1099.259,309.502,-81.984,178.754,18.069,152.125
C09903=1099.264,309.751,-82.016,178.758,18.071,152.125
C09904=1099.270,309.999,-82.046,178.761,18.074,152.125
C09905=1099.276,310.246,-82.078,178.764,18.076,152.125
C09906=1099.281,310.495,-82.109,178.768,18.078,152.124
C09907=1099.287,310.742,-82.140,178.771,18.080,152.124
C09908=1099.293,310.990,-82.171,178.774,18.083,152.124
C09909=1099.299,311.238,-82.203,178.778,18.085,152.124
C09910=1099.304,311.486,-82.233,178.781,18.087,152.124
C09911=1099.310,311.734,-82.265,178.784,18.090,152.124
C09912=1099.316,311.982,-82.296,178.787,18.091,152.124
C09913=1099.322,312.230,-82.327,178.791,18.094,152.124
C09914=1099.328,312.478,-82.360,178.794,18.096,152.124
C09915=1099.333,312.726,-82.390,178.797,18.099,152.124
C09916=1099.339,312.973,-82.422,178.801,18.100,152.123
C09917=1099.344,313.222,-82.453,178.804,18.103,152.123
C09918=1099.351,313.469,-82.484,178.807,18.105,152.123
C09919=1099.357,313.718,-82.516,178.810,18.108,152.123
C09920=1099.362,313.966,-82.547,178.814,18.110,152.123
C09921=1099.368,314.214,-82.578,178.817,18.112,152.123
C09922=1099.374,314.461,-82.610,178.820,18.114,152.123
C09923=1099.379,314.710,-82.641,178.823,18.117,152.123
C09924=1099.386,314.957,-82.672,178.827,18.119,152.123
C09925=1099.392,315.205,-82.704,178.830,18.121,152.123
C09926=1099.397,315.453,-82.736,178.833,18.123,152.123
C09927=1099.402,315.701,-82.767,178.836,18.126,152.123
C09928=1099.411,316.087,-82.817,178.842,18.130,152.122
C09929=1099.419,316.473,-82.866,178.846,18.134,152.123
C09930=1099.428,316.860,-82.915,178.852,18.138,152.122
C09931=1099.437,317.246,-82.964,178.857,18.142,152.122
C09932=1099.443,317.493,-82.996,178.860,18.144,152.122
C09933=1099.449,317.741,-83.028,178.863,18.146,152.122
C09934=1099.454,317.989,-83.060,178.867,18.149,152.122
C09935=1099.458,318.237,-83.091,178.869,18.151,152.122
C09936=1099.464,318.486,-83.123,178.873,18.154,152.122
C09937=1099.470,318.733,-83.155,178.876,18.156,152.122
C09938=1099.476,318.981,-83.187,178.880,18.159,152.122
C09939=1099.481,319.229,-83.219,178.883,18.161,152.122
C09940=1099.487,319.477,-83.251,178.886,18.164,152.122
C09941=1099.493,319.725,-83.282,178.889,18.167,152.122
C09942=1099.499,319.973,-83.314,178.892,18.169,152.122
C09943=1099.504,320.220,-83.346,178.896,18.171,152.122
C09944=1099.510,320.468,-83.378,178.899,18.174,152.122
C09945=1099.515,320.716,-83.410,178.902,18.177,152.122
C09946=1099.521,320.964,-83.442,178.905,18.179,152.122
C09947=1099.526,321.212,-83.474,178.909,18.182,152.122
C09948=1099.532,321.460,-83.506,178.912,18.184,152.122
C09949=1099.537,321.708,-83.538,178.915,18.187,152.122
C09950=1099.543,321.956,-83.570,178.918,18.189,152.122
C09951=1099.550,322.204,-83.603,178.922,18.192,152.122
C09952=1099.555,322.451,-83.634,178.925,18.194,152.122
C09953=1099.560,322.700,-83.667,178.928,18.197,152.122
C09954=1099.566,322.947,-83.699,178.931,18.199,152.122
C09955=1099.572,323.195,-83.731,178.935,18.202,152.122
C09956=1099.578,323.444,-83.763,178.938,18.205,152.122
C09957=1099.583,323.690,-83.795,178.941,18.207,152.122
C09958=1099.589,323.939,-83.827,178.944,18.210,152.122
C09959=1099.594,324.186,-83.859,178.947,18.213,152.122
C09960=1099.600,324.435,-83.891,178.950,18.215,152.122
C09961=1099.606,324.682,-83.924,178.954,18.217,152.122
C09962=1099.612,324.930,-83.956,178.957,18.221,152.122
C09963=1099.618,325.178,-83.988,178.961,18.223,152.122
C09964=1099.623,325.427,-84.020,178.964,18.226,152.122
C09965=1099.629,325.673,-84.053,178.967,18.228,152.122
C09966=1099.635,325.922,-84.085,178.970,18.231,152.122
C09967=1099.641,326.169,-84.117,178.973,18.233,152.122
C09968=1099.645,326.417,-84.150,178.977,18.236,152.122
C09969=1099.651,326.665,-84.182,178.980,18.239,152.122
C09970=1099.658,326.913,-84.214,178.983,18.242,152.122
C09971=1099.663,327.161,-84.247,178.986,18.244,152.122
C09972=1099.669,327.408,-84.279,178.989,18.247,152.122
C09973=1099.675,327.656,-84.312,178.992,18.250,152.122
C09974=1099.681,327.905,-84.344,178.996,18.253,152.122
C09975=1099.686,328.153,-84.377,178.999,18.255,152.122
C09976=1099.692,328.400,-84.409,179.002,18.258,152.122
C09977=1099.698,328.648,-84.441,179.005,18.260,152.122
C09978=1099.703,328.896,-84.474,179.009,18.263,152.122
C09979=1099.709,329.144,-84.507,179.012,18.266,152.122
C09980=1099.718,329.523,-84.556,179.017,18.270,152.122
C09981=1099.726,329.902,-84.606,179.022,18.274,152.123
C09982=1099.736,330.281,-84.655,179.027,18.278,152.123
C09983=1099.745,330.660,-84.706,179.032,18.282,152.123
C09984=1099.750,330.908,-84.739,179.035,18.286,152.123
C09985=1099.756,331.156,-84.771,179.038,18.288,152.123
C09986=1099.762,331.403,-84.804,179.041,18.291,152.123
C09987=1099.767,331.651,-84.837,179.044,18.294,152.123
C09988=1099.773,331.899,-84.869,179.048,18.296,152.123
C09989=1099.779,332.147,-84.902,179.051,18.299,152.123
C09990=1099.785,332.394,-84.935,179.054,18.302,152.123
C09991=1099.791,332.642,-84.968,179.057,18.305,152.123
C09992=1099.797,332.890,-85.000,179.060,18.307,152.123
C09993=1099.802,333.138,-85.033,179.064,18.311,152.123
C09994=1099.808,333.385,-85.066,179.067,18.314,152.123
C09995=1099.814,333.633,-85.099,179.070,18.316,152.124
C09996=1099.819,333.882,-85.132,179.073,18.319,152.124
//INST
///DATE 2021/06/17 10:53
///ATTR SC,RW,RJ
////FRAME ROBOT
///GROUP1 RB1
NOP
MOVL C00000 V=800.0 PL=0
MOVL C00001 V=800.0 PL=0
MOVL C00002 V=800.0 PL=0
MOVL C00003 V=800.0 PL=0
MOVL C00004 V=800.0 PL=0
MOVL C00005 V=800.0 PL=0
MOVL C00006 V=800.0 PL=0
MOVL C00007 V=800.0 PL=0
MOVL C00008 V=800.0 PL=0
MOVL C00009 V=800.0 PL=0
MOVL C00010 V=800.0 PL=0
MOVL C00011 V=800.0 PL=0
MOVL C00012 V=800.0 PL=0
MOVL C00013 V=800.0 PL=0
MOVL C00014 V=800.0 PL=0
MOVL C00015 V=800.0 PL=0
MOVL C00016 V=800.0 PL=0
MOVL C00017 V=800.0 PL=0
MOVL C00018 V=800.0 PL=0
MOVL C00019 V=800.0 PL=0
MOVL C00020 V=800.0 PL=0
MOVL C00021 V=800.0 PL=0
MOVL C00022 V=800.0 PL=0
MOVL C00023 V=800.0 PL=0
MOVL C00024 V=800.0 PL=0
MOVL C00025 V=800.0 PL=0
MOVL C00026 V=800.0 PL=0
MOVL C00027 V=800.0 PL=0
MOVL C00028 V=800.0 PL=0
MOVL C00029 V=800.0 PL=0
MOVL C00030 V=800.0 PL=0
MOVL C00031 V=800.0 PL=0
MOVL C00032 V=800.0 PL=0
MOVL C00033 V=800.0 PL=0
MOVL C00034 V=800.0 PL=0
MOVL C00035 V=800.0 PL=0
MOVL C00036 V=800.0 PL=0
MOVL C00037 V=800.0 PL=0
MOVL C00038 V=800.0 PL=0
MOVL C00039 V=800.0 PL=0
MOVL C00040 V=800.0 PL=0
MOVL C00041 V=800.0 PL=0
MOVL C00042 V=800.0 PL=0
MOVL C00043 V=800.0 PL=0
MOVL C00044 V=800.0 PL=0
MOVL C00045 V=800.0 PL=0
MOVL C00046 V=800.0 PL=0
MOVL C00047 V=800.0 PL=0
MOVL C00048 V=800.0 PL=0
MOVL C00049 V=800.0 PL=0
MOVL C00050 V=800.0 PL=0
MOVL C00051 V=800.0 PL=0
MOVL C00052 V=800.0 PL=0
MOVL C00053 V=800.0 PL=0
MOVL C00054 V=800.0 PL=0
MOVL C00055 V=800.0 PL=0
MOVL C00056 V=800.0 PL=0
MOVL C00057 V=800.0 PL=0
MOVL C00058 V=800.0 PL=0
MOVL C00059 V=800.0 PL=0
MOVL C00060 V=800.0 PL=0
MOVL C00061 V=800.0 PL=0
MOVL C00062 V=800.0 PL=0
MOVL C00063 V=800.0 PL=0
MOVL C00064 V=800.0 PL=0
MOVL C00065 V=800.0 PL=0
MOVL C00066 V=800.0 PL=0
MOVL C00067 V=800.0 PL=0
MOVL C00068 V=800.0 PL=0
MOVL C00069 V=800.0 PL=0
MOVL C00070 V=800.0 PL=0
MOVL C00071 V=800.0 PL=0
MOVL C00072 V=800.0 PL=0
MOVL C00073 V=800.0 PL=0
MOVL C00074 V=800.0 PL=0
MOVL C00075 V=800.0 PL=0
MOVL C00076 V=800.0 PL=0
MOVL C00077 V=800.0 PL=0
MOVL C00078 V=800.0 PL=0
MOVL C00079 V=800.0 PL=0
MOVL C00080 V=800.0 PL=0
MOVL C00081 V=800.0 PL=0
MOVL C00082 V=800.0 PL=0
MOVL C00083 V=800.0 PL=0
MOVL C00084 V=800.0 PL=0
MOVL C00085 V=800.0 PL=0
MOVL C00086 V=800.0 PL=0
MOVL C00087 V=800.0 PL=0
MOVL C00088 V=800.0 PL=0
MOVL C00089 V=800.0 PL=0
MOVL C00090 V=800.0 PL=0
MOVL C00091 V=800.0 PL=0
MOVL C00092 V=800.0 PL=0
MOVL C00093 V=800.0 PL=0
MOVL C00094 V=800.0 PL=0
MOVL C00095 V=800.0 PL=0
MOVL C00096 V=800.0 PL=0
MOVL C00097 V=800.0 PL=0
MOVL C00098 V=800.0 PL=0
MOVL C00099 V=800.0 PL=0
MOVL C00100 V=800.0 PL=0
MOVL C00101 V=800.0 PL=0
MOVL C00102 V=800.0 PL=0
MOVL C00103 V=800.0 PL=0
MOVL C00104 V=800.0 PL=0
MOVL C00105 V=800.0 PL=0
MOVL C00106 V=800.0 PL=0
MOVL C00107 V=800.0 PL=0
MOVL C00108 V=800.0 PL=0
MOVL C00109 V=800.0 PL=0
MOVL C00110 V=800.0 PL=0
MOVL C00111 V=800.0 PL=0
MOVL C00112 V=800.0 PL=0
MOVL C00113 V=800.0 PL=0
MOVL C00114 V=800.0 PL=0
MOVL C00115 V=800.0 PL=0
MOVL C00116 V=800.0 PL=0
MOVL C00117 V=800.0 PL=0
MOVL C00118 V=800.0 PL=0
MOVL C00119 V=800.0 PL=0
MOVL C00120 V=800.0 PL=0
MOVL C00121 V=800.0 PL=0
MOVL C00122 V=800.0 PL=0
MOVL C00123 V=800.0 PL=0
MOVL C00124 V=800.0 PL=0
MOVL C00125 V=800.0 PL=0
MOVL C00126 V=800.0 PL=0
MOVL C00127 V=800.0 PL=0
MOVL C00128 V=800.0 PL=0
MOVL C00129 V=800.0 PL=0
MOVL C00130 V=800.0 PL=0
MOVL C00131 V=800.0 PL=0
MOVL C00132 V=800.0 PL=0
MOVL C00133 V=800.0 PL=0
MOVL C00134 V=800.0 PL=0
MOVL C00135 V=800.0 PL=0
MOVL C00136 V=800.0 PL=0
MOVL C00137 V=800.0 PL=0
MOVL C00138 V=800.0 PL=0
MOVL C00139 V=800.0 PL=0
MOVL C00140 V=800.0 PL=0
MOVL C00141 V=800.0 PL=0
MOVL C00142 V=800.0 PL=0
MOVL C00143 V=800.0 PL=0
MOVL C00144 V=800.0 PL=0
MOVL C00145 V=800.0 PL=0
MOVL C00146 V=800.0 PL=0
MOVL C00147 V=800.0 PL=0
MOVL C00148 V=800.0 PL=0
MOVL C00149 V=800.0 PL=0
MOVL C00150 V=800.0 PL=0
MOVL C00151 V=800.0 PL=0
MOVL C00152 V=800.0 PL=0
MOVL C00153 V=800.0 PL=0
MOVL C00154 V=800.0 PL=0
MOVL C00155 V=800.0 PL=0
MOVL C00156 V=800.0 PL=0
MOVL C00157 V=800.0 PL=0
MOVL C00158 V=800.0 PL=0
MOVL C00159 V=800.0 PL=0
MOVL C00160 V=800.0 PL=0
MOVL C00161 V=800.0 PL=0
MOVL C00162 V=800.0 PL=0
MOVL C00163 V=800.0 PL=0
MOVL C00164 V=800.0 PL=0
MOVL C00165 V=800.0 PL=0
MOVL C00166 V=800.0 PL=0
MOVL C00167 V=800.0 PL=0
MOVL C00168 V=800.0 PL=0
MOVL C00169 V=800.0 PL=0
MOVL C00170 V=800.0 PL=0
MOVL C00171 V=800.0 PL=0
MOVL C00172 V=800.0 PL=0
MOVL C00173 V=800.0 PL=0
MOVL C00174 V=800.0 PL=0
MOVL C00175 V=800.0 PL=0
MOVL C00176 V=800.0 PL=0
MOVL C00177 V=800.0 PL=0
MOVL C00178 V=800.0 PL=0
MOVL C00179 V=800.0 PL=0
MOVL C00180 V=800.0 PL=0
MOVL C00181 V=800.0 PL=0
MOVL C00182 V=800.0 PL=0
MOVL C00183 V=800.0 PL=0
MOVL C00184 V=800.0 PL=0
MOVL C00185 V=800.0 PL=0
MOVL C00186 V=800.0 PL=0
MOVL C00187 V=800.0 PL=0
MOVL C00188 V=800.0 PL=0
MOVL C00189 V=800.0 PL=0
MOVL C00190 V=800.0 PL=0
MOVL C00191 V=800.0 PL=0
MOVL C00192 V=800.0 PL=0
MOVL C00193 V=800.0 PL=0
MOVL C00194 V=800.0 PL=0
MOVL C00195 V=800.0 PL=0
MOVL C00196 V=800.0 PL=0
MOVL C00197 V=800.0 PL=0
MOVL C00198 V=800.0 PL=0
MOVL C00199 V=800.0 PL=0
MOVL C00200 V=800.0 PL=0
MOVL C00201 V=800.0 PL=0
MOVL C00202 V=800.0 PL=0
MOVL C00203 V=800.0 PL=0
MOVL C00204 V=800.0 PL=0
MOVL C00205 V=800.0 PL=0
MOVL C00206 V=800.0 PL=0
MOVL C00207 V=800.0 PL=0
MOVL C00208 V=800.0 PL=0
MOVL C00209 V=800.0 PL=0
MOVL C00210 V=800.0 PL=0
MOVL C00211 V=800.0 PL=0
MOVL C00212 V=800.0 PL=0
MOVL C00213 V=800.0 PL=0
MOVL C00214 V=800.0 PL=0
MOVL C00215 V=800.0 PL=0
MOVL C00216 V=800.0 PL=0
MOVL C00217 V=800.0 PL=0
MOVL C00218 V=800.0 PL=0
MOVL C00219 V=800.0 PL=0
MOVL C00220 V=800.0 PL=0
MOVL C00221 V=800.0 PL=0
MOVL C00222 V=800.0 PL=0
MOVL C00223 V=800.0 PL=0
MOVL C00224 V=800.0 PL=0
MOVL C00225 V=800.0 PL=0
MOVL C00226 V=800.0 PL=0
MOVL C00227 V=800.0 PL=0
MOVL C00228 V=800.0 PL=0
MOVL C00229 V=800.0 PL=0
MOVL C00230 V=800.0 PL=0
MOVL C00231 V=800.0 PL=0
MOVL C00232 V=800.0 PL=0
MOVL C00233 V=800.0 PL=0
MOVL C00234 V=800.0 PL=0
MOVL C00235 V=800.0 PL=0
MOVL C00236 V=800.0 PL=0
MOVL C00237 V=800.0 PL=0
MOVL C00238 V=800.0 PL=0
MOVL C00239 V=800.0 PL=0
MOVL C00240 V=800.0 PL=0
MOVL C00241 V=800.0 PL=0
MOVL C00242 V=800.0 PL=0
MOVL C00243 V=800.0 PL=0
MOVL C00244 V=800.0 PL=0
MOVL C00245 V=800.0 PL=0
MOVL C00246 V=800.0 PL=0
MOVL C00247 V=800.0 PL=0
MOVL C00248 V=800.0 PL=0
MOVL C00249 V=800.0 PL=0
MOVL C00250 V=800.0 PL=0
MOVL C00251 V=800.0 PL=0
MOVL C00252 V=800.0 PL=0
MOVL C00253 V=800.0 PL=0
MOVL C00254 V=800.0 PL=0
MOVL C00255 V=800.0 PL=0
MOVL C00256 V=800.0 PL=0
MOVL C00257 V=800.0 PL=0
MOVL C00258 V=800.0 PL=0
MOVL C00259 V=800.0 PL=0
MOVL C00260 V=800.0 PL=0
MOVL C00261 V=800.0 PL=0
MOVL C00262 V=800.0 PL=0
MOVL C00263 V=800.0 PL=0
MOVL C00264 V=800.0 PL=0
MOVL C00265 V=800.0 PL=0
MOVL C00266 V=800.0 PL=0
MOVL C00267 V=800.0 PL=0
MOVL C00268 V=800.0 PL=0
MOVL C00269 V=800.0 PL=0
MOVL C00270 V=800.0 PL=0
MOVL C00271 V=800.0 PL=0
MOVL C00272 V=800.0 PL=0
MOVL C00273 V=800.0 PL=0
MOVL C00274 V=800.0 PL=0
MOVL C00275 V=800.0 PL=0
MOVL C00276 V=800.0 PL=0
MOVL C00277 V=800.0 PL=0
MOVL C00278 V=800.0 PL=0
MOVL C00279 V=800.0 PL=0
MOVL C00280 V=800.0 PL=0
MOVL C00281 V=800.0 PL=0
MOVL C00282 V=800.0 PL=0
MOVL C00283 V=800.0 PL=0
MOVL C00284 V=800.0 PL=0
MOVL C00285 V=800.0 PL=0
MOVL C00286 V=800.0 PL=0
MOVL C00287 V=800.0 PL=0
MOVL C00288 V=800.0 PL=0
MOVL C00289 V=800.0 PL=0
MOVL C00290 V=800.0 PL=0
MOVL C00291 V=800.0 PL=0
MOVL C00292 V=800.0 PL=0
MOVL C00293 V=800.0 PL=0
MOVL C00294 V=800.0 PL=0
MOVL C00295 V=800.0 PL=0
MOVL C00296 V=800.0 PL=0
MOVL C00297 V=800.0 PL=0
MOVL C00298 V=800.0 PL=0
MOVL C00299 V=800.0 PL=0
MOVL C00300 V=800.0 PL=0
MOVL C00301 V=800.0 PL=0
MOVL C00302 V=800.0 PL=0
MOVL C00303 V=800.0 PL=0
MOVL C00304 V=800.0 PL=0
MOVL C00305 V=800.0 PL=0
MOVL C00306 V=800.0 PL=0
MOVL C00307 V=800.0 PL=0
MOVL C00308 V=800.0 PL=0
MOVL C00309 V=800.0 PL=0
MOVL C00310 V=800.0 PL=0
MOVL C00311 V=800.0 PL=0
MOVL C00312 V=800.0 PL=0
MOVL C00313 V=800.0 PL=0
MOVL C00314 V=800.0 PL=0
MOVL C00315 V=800.0 PL=0
MOVL C00316 V=800.0 PL=0
MOVL C00317 V=800.0 PL=0
MOVL C00318 V=800.0 PL=0
MOVL C00319 V=800.0 PL=0
MOVL C00320 V=800.0 PL=0
MOVL C00321 V=800.0 PL=0
MOVL C00322 V=800.0 PL=0
MOVL C00323 V=800.0 PL=0
MOVL C00324 V=800.0 PL=0
MOVL C00325 V=800.0 PL=0
MOVL C00326 V=800.0 PL=0
MOVL C00327 V=800.0 PL=0
MOVL C00328 V=800.0 PL=0
MOVL C00329 V=800.0 PL=0
MOVL C00330 V=800.0 PL=0
MOVL C00331 V=800.0 PL=0
MOVL C00332 V=800.0 PL=0
MOVL C00333 V=800.0 PL=0
MOVL C00334 V=800.0 PL=0
MOVL C00335 V=800.0 PL=0
MOVL C00336 V=800.0 PL=0
MOVL C00337 V=800.0 PL=0
MOVL C00338 V=800.0 PL=0
MOVL C00339 V=800.0 PL=0
MOVL C00340 V=800.0 PL=0
MOVL C00341 V=800.0 PL=0
MOVL C00342 V=800.0 PL=0
MOVL C00343 V=800.0 PL=0
MOVL C00344 V=800.0 PL=0
MOVL C00345 V=800.0 PL=0
MOVL C00346 V=800.0 PL=0
MOVL C00347 V=800.0 PL=0
MOVL C00348 V=800.0 PL=0
MOVL C00349 V=800.0 PL=0
MOVL C00350 V=800.0 PL=0
MOVL C00351 V=800.0 PL=0
MOVL C00352 V=800.0 PL=0
MOVL C00353 V=800.0 PL=0
MOVL C00354 V=800.0 PL=0
MOVL C00355 V=800.0 PL=0
MOVL C00356 V=800.0 PL=0
MOVL C00357 V=800.0 PL=0
MOVL C00358 V=800.0 PL=0
MOVL C00359 V=800.0 PL=0
MOVL C00360 V=800.0 PL=0
MOVL C00361 V=800.0 PL=0
MOVL C00362 V=800.0 PL=0
MOVL C00363 V=800.0 PL=0
MOVL C00364 V=800.0 PL=0
MOVL C00365 V=800.0 PL=0
MOVL C00366 V=800.0 PL=0
MOVL C00367 V=800.0 PL=0
MOVL C00368 V=800.0 PL=0
MOVL C00369 V=800.0 PL=0
MOVL C00370 V=800.0 PL=0
MOVL C00371 V=800.0 PL=0
MOVL C00372 V=800.0 PL=0
MOVL C00373 V=800.0 PL=0
MOVL C00374 V=800.0 PL=0
MOVL C00375 V=800.0 PL=0
MOVL C00376 V=800.0 PL=0
MOVL C00377 V=800.0 PL=0
MOVL C00378 V=800.0 PL=0
MOVL C00379 V=800.0 PL=0
MOVL C00380 V=800.0 PL=0
MOVL C00381 V=800.0 PL=0
MOVL C00382 V=800.0 PL=0
MOVL C00383 V=800.0 PL=0
MOVL C00384 V=800.0 PL=0
MOVL C00385 V=800.0 PL=0
MOVL C00386 V=800.0 PL=0
MOVL C00387 V=800.0 PL=0
MOVL C00388 V=800.0 PL=0
MOVL C00389 V=800.0 PL=0
MOVL C00390 V=800.0 PL=0
MOVL C00391 V=800.0 PL=0
MOVL C00392 V=800.0 PL=0
MOVL C00393 V=800.0 PL=0
MOVL C00394 V=800.0 PL=0
MOVL C00395 V=800.0 PL=0
MOVL C00396 V=800.0 PL=0
MOVL C00397 V=800.0 PL=0
MOVL C00398 V=800.0 PL=0
MOVL C00399 V=800.0 PL=0
MOVL C00400 V=800.0 PL=0
MOVL C00401 V=800.0 PL=0
MOVL C00402 V=800.0 PL=0
MOVL C00403 V=800.0 PL=0
MOVL C00404 V=800.0 PL=0
MOVL C00405 V=800.0 PL=0
MOVL C00406 V=800.0 PL=0
MOVL C00407 V=800.0 PL=0
MOVL C00408 V=800.0 PL=0
MOVL C00409 V=800.0 PL=0
MOVL C00410 V=800.0 PL=0
MOVL C00411 V=800.0 PL=0
MOVL C00412 V=800.0 PL=0
MOVL C00413 V=800.0 PL=0
MOVL C00414 V=800.0 PL=0
MOVL C00415 V=800.0 PL=0
MOVL C00416 V=800.0 PL=0
MOVL C00417 V=800.0 PL=0
MOVL C00418 V=800.0 PL=0
MOVL C00419 V=800.0 PL=0
MOVL C00420 V=800.0 PL=0
MOVL C00421 V=800.0 PL=0
MOVL C00422 V=800.0 PL=0
MOVL C00423 V=800.0 PL=0
MOVL C00424 V=800.0 PL=0
MOVL C00425 V=800.0 PL=0
MOVL C00426 V=800.0 PL=0
MOVL C00427 V=800.0 PL=0
MOVL C00428 V=800.0 PL=0
MOVL C00429 V=800.0 PL=0
MOVL C00430 V=800.0 PL=0
MOVL C00431 V=800.0 PL=0
MOVL C00432 V=800.0 PL=0
MOVL C00433 V=800.0 PL=0
MOVL C00434 V=800.0 PL=0
MOVL C00435 V=800.0 PL=0
MOVL C00436 V=800.0 PL=0
MOVL C00437 V=800.0 PL=0
MOVL C00438 V=800.0 PL=0
MOVL C00439 V=800.0 PL=0
MOVL C00440 V=800.0 PL=0
MOVL C00441 V=800.0 PL=0
MOVL C00442 V=800.0 PL=0
MOVL C00443 V=800.0 PL=0
MOVL C00444 V=800.0 PL=0
MOVL C00445 V=800.0 PL=0
MOVL C00446 V=800.0 PL=0
MOVL C00447 V=800.0 PL=0
MOVL C00448 V=800.0 PL=0
MOVL C00449 V=800.0 PL=0
MOVL C00450 V=800.0 PL=0
MOVL C00451 V=800.0 PL=0
MOVL C00452 V=800.0 PL=0
MOVL C00453 V=800.0 PL=0
MOVL C00454 V=800.0 PL=0
MOVL C00455 V=800.0 PL=0
MOVL C00456 V=800.0 PL=0
MOVL C00457 V=800.0 PL=0
MOVL C00458 V=800.0 PL=0
MOVL C00459 V=800.0 PL=0
MOVL C00460 V=800.0 PL=0
MOVL C00461 V=800.0 PL=0
MOVL C00462 V=800.0 PL=0
MOVL C00463 V=800.0 PL=0
MOVL C00464 V=800.0 PL=0
MOVL C00465 V=800.0 PL=0
MOVL C00466 V=800.0 PL=0
MOVL C00467 V=800.0 PL=0
MOVL C00468 V=800.0 PL=0
MOVL C00469 V=800.0 PL=0
MOVL C00470 V=800.0 PL=0
MOVL C00471 V=800.0 PL=0
MOVL C00472 V=800.0 PL=0
MOVL C00473 V=800.0 PL=0
MOVL C00474 V=800.0 PL=0
MOVL C00475 V=800.0 PL=0
MOVL C00476 V=800.0 PL=0
MOVL C00477 V=800.0 PL=0
MOVL C00478 V=800.0 PL=0
MOVL C00479 V=800.0 PL=0
MOVL C00480 V=800.0 PL=0
MOVL C00481 V=800.0 PL=0
MOVL C00482 V=800.0 PL=0
MOVL C00483 V=800.0 PL=0
MOVL C00484 V=800.0 PL=0
MOVL C00485 V=800.0 PL=0
MOVL C00486 V=800.0 PL=0
MOVL C00487 V=800.0 PL=0
MOVL C00488 V=800.0 PL=0
MOVL C00489 V=800.0 PL=0
MOVL C00490 V=800.0 PL=0
MOVL C00491 V=800.0 PL=0
MOVL C00492 V=800.0 PL=0
MOVL C00493 V=800.0 PL=0
MOVL C00494 V=800.0 PL=0
MOVL C00495 V=800.0 PL=0
MOVL C00496 V=800.0 PL=0
MOVL C00497 V=800.0 PL=0
MOVL C00498 V=800.0 PL=0
MOVL C00499 V=800.0 PL=0
MOVL C00500 V=800.0 PL=0
MOVL C00501 V=800.0 PL=0
MOVL C00502 V=800.0 PL=0
MOVL C00503 V=800.0 PL=0
MOVL C00504 V=800.0 PL=0
MOVL C00505 V=800.0 PL=0
MOVL C00506 V=800.0 PL=0
MOVL C00507 V=800.0 PL=0
MOVL C00508 V=800.0 PL=0
MOVL C00509 V=800.0 PL=0
MOVL C00510 V=800.0 PL=0
MOVL C00511 V=800.0 PL=0
MOVL C00512 V=800.0 PL=0
MOVL C00513 V=800.0 PL=0
MOVL C00514 V=800.0 PL=0
MOVL C00515 V=800.0 PL=0
MOVL C00516 V=800.0 PL=0
MOVL C00517 V=800.0 PL=0
MOVL C00518 V=800.0 PL=0
MOVL C00519 V=800.0 PL=0
MOVL C00520 V=800.0 PL=0
MOVL C00521 V=800.0 PL=0
MOVL C00522 V=800.0 PL=0
MOVL C00523 V=800.0 PL=0
MOVL C00524 V=800.0 PL=0
MOVL C00525 V=800.0 PL=0
MOVL C00526 V=800.0 PL=0
MOVL C00527 V=800.0 PL=0
MOVL C00528 V=800.0 PL=0
MOVL C00529 V=800.0 PL=0
MOVL C00530 V=800.0 PL=0
MOVL C00531 V=800.0 PL=0
MOVL C00532 V=800.0 PL=0
MOVL C00533 V=800.0 PL=0
MOVL C00534 V=800.0 PL=0
MOVL C00535 V=800.0 PL=0
MOVL C00536 V=800.0 PL=0
MOVL C00537 V=800.0 PL=0
MOVL C00538 V=800.0 PL=0
MOVL C00539 V=800.0 PL=0
MOVL C00540 V=800.0 PL=0
MOVL C00541 V=800.0 PL=0
MOVL C00542 V=800.0 PL=0
MOVL C00543 V=800.0 PL=0
MOVL C00544 V=800.0 PL=0
MOVL C00545 V=800.0 PL=0
MOVL C00546 V=800.0 PL=0
MOVL C00547 V=800.0 PL=0
MOVL C00548 V=800.0 PL=0
MOVL C00549 V=800.0 PL=0
MOVL C00550 V=800.0 PL=0
MOVL C00551 V=800.0 PL=0
MOVL C00552 V=800.0 PL=0
MOVL C00553 V=800.0 PL=0
MOVL C00554 V=800.0 PL=0
MOVL C00555 V=800.0 PL=0
MOVL C00556 V=800.0 PL=0
MOVL C00557 V=800.0 PL=0
MOVL C00558 V=800.0 PL=0
MOVL C00559 V=800.0 PL=0
MOVL C00560 V=800.0 PL=0
MOVL C00561 V=800.0 PL=0
MOVL C00562 V=800.0 PL=0
MOVL C00563 V=800.0 PL=0
MOVL C00564 V=800.0 PL=0
MOVL C00565 V=800.0 PL=0
MOVL C00566 V=800.0 PL=0
MOVL C00567 V=800.0 PL=0
MOVL C00568 V=800.0 PL=0
MOVL C00569 V=800.0 PL=0
MOVL C00570 V=800.0 PL=0
MOVL C00571 V=800.0 PL=0
MOVL C00572 V=800.0 PL=0
MOVL C00573 V=800.0 PL=0
MOVL C00574 V=800.0 PL=0
MOVL C00575 V=800.0 PL=0
MOVL C00576 V=800.0 PL=0
MOVL C00577 V=800.0 PL=0
MOVL C00578 V=800.0 PL=0
MOVL C00579 V=800.0 PL=0
MOVL C00580 V=800.0 PL=0
MOVL C00581 V=800.0 PL=0
MOVL C00582 V=800.0 PL=0
MOVL C00583 V=800.0 PL=0
MOVL C00584 V=800.0 PL=0
MOVL C00585 V=800.0 PL=0
MOVL C00586 V=800.0 PL=0
MOVL C00587 V=800.0 PL=0
MOVL C00588 V=800.0 PL=0
MOVL C00589 V=800.0 PL=0
MOVL C00590 V=800.0 PL=0
MOVL C00591 V=800.0 PL=0
MOVL C00592 V=800.0 PL=0
MOVL C00593 V=800.0 PL=0
MOVL C00594 V=800.0 PL=0
MOVL C00595 V=800.0 PL=0
MOVL C00596 V=800.0 PL=0
MOVL C00597 V=800.0 PL=0
MOVL C00598 V=800.0 PL=0
MOVL C00599 V=800.0 PL=0
MOVL C00600 V=800.0 PL=0
MOVL C00601 V=800.0 PL=0
MOVL C00602 V=800.0 PL=0
MOVL C00603 V=800.0 PL=0
MOVL C00604 V=800.0 PL=0
MOVL C00605 V=800.0 PL=0
MOVL C00606 V=800.0 PL=0
MOVL C00607 V=800.0 PL=0
MOVL C00608 V=800.0 PL=0
MOVL C00609 V=800.0 PL=0
MOVL C00610 V=800.0 PL=0
MOVL C00611 V=800.0 PL=0
MOVL C00612 V=800.0 PL=0
MOVL C00613 V=800.0 PL=0
MOVL C00614 V=800.0 PL=0
MOVL C00615 V=800.0 PL=0
MOVL C00616 V=800.0 PL=0
MOVL C00617 V=800.0 PL=0
MOVL C00618 V=800.0 PL=0
MOVL C00619 V=800.0 PL=0
MOVL C00620 V=800.0 PL=0
MOVL C00621 V=800.0 PL=0
MOVL C00622 V=800.0 PL=0
MOVL C00623 V=800.0 PL=0
MOVL C00624 V=800.0 PL=0
MOVL C00625 V=800.0 PL=0
MOVL C00626 V=800.0 PL=0
MOVL C00627 V=800.0 PL=0
MOVL C00628 V=800.0 PL=0
MOVL C00629 V=800.0 PL=0
MOVL C00630 V=800.0 PL=0
MOVL C00631 V=800.0 PL=0
MOVL C00632 V=800.0 PL=0
MOVL C00633 V=800.0 PL=0
MOVL C00634 V=800.0 PL=0
MOVL C00635 V=800.0 PL=0
MOVL C00636 V=800.0 PL=0
MOVL C00637 V=800.0 PL=0
MOVL C00638 V=800.0 PL=0
MOVL C00639 V=800.0 PL=0
MOVL C00640 V=800.0 PL=0
MOVL C00641 V=800.0 PL=0
MOVL C00642 V=800.0 PL=0
MOVL C00643 V=800.0 PL=0
MOVL C00644 V=800.0 PL=0
MOVL C00645 V=800.0 PL=0
MOVL C00646 V=800.0 PL=0
MOVL C00647 V=800.0 PL=0
MOVL C00648 V=800.0 PL=0
MOVL C00649 V=800.0 PL=0
MOVL C00650 V=800.0 PL=0
MOVL C00651 V=800.0 PL=0
MOVL C00652 V=800.0 PL=0
MOVL C00653 V=800.0 PL=0
MOVL C00654 V=800.0 PL=0
MOVL C00655 V=800.0 PL=0
MOVL C00656 V=800.0 PL=0
MOVL C00657 V=800.0 PL=0
MOVL C00658 V=800.0 PL=0
MOVL C00659 V=800.0 PL=0
MOVL C00660 V=800.0 PL=0
MOVL C00661 V=800.0 PL=0
MOVL C00662 V=800.0 PL=0
MOVL C00663 V=800.0 PL=0
MOVL C00664 V=800.0 PL=0
MOVL C00665 V=800.0 PL=0
MOVL C00666 V=800.0 PL=0
MOVL C00667 V=800.0 PL=0
MOVL C00668 V=800.0 PL=0
MOVL C00669 V=800.0 PL=0
MOVL C00670 V=800.0 PL=0
MOVL C00671 V=800.0 PL=0
MOVL C00672 V=800.0 PL=0
MOVL C00673 V=800.0 PL=0
MOVL C00674 V=800.0 PL=0
MOVL C00675 V=800.0 PL=0
MOVL C00676 V=800.0 PL=0
MOVL C00677 V=800.0 PL=0
MOVL C00678 V=800.0 PL=0
MOVL C00679 V=800.0 PL=0
MOVL C00680 V=800.0 PL=0
MOVL C00681 V=800.0 PL=0
MOVL C00682 V=800.0 PL=0
MOVL C00683 V=800.0 PL=0
MOVL C00684 V=800.0 PL=0
MOVL C00685 V=800.0 PL=0
MOVL C00686 V=800.0 PL=0
MOVL C00687 V=800.0 PL=0
MOVL C00688 V=800.0 PL=0
MOVL C00689 V=800.0 PL=0
MOVL C00690 V=800.0 PL=0
MOVL C00691 V=800.0 PL=0
MOVL C00692 V=800.0 PL=0
MOVL C00693 V=800.0 PL=0
MOVL C00694 V=800.0 PL=0
MOVL C00695 V=800.0 PL=0
MOVL C00696 V=800.0 PL=0
MOVL C00697 V=800.0 PL=0
MOVL C00698 V=800.0 PL=0
MOVL C00699 V=800.0 PL=0
MOVL C00700 V=800.0 PL=0
MOVL C00701 V=800.0 PL=0
MOVL C00702 V=800.0 PL=0
MOVL C00703 V=800.0 PL=0
MOVL C00704 V=800.0 PL=0
MOVL C00705 V=800.0 PL=0
MOVL C00706 V=800.0 PL=0
MOVL C00707 V=800.0 PL=0
MOVL C00708 V=800.0 PL=0
MOVL C00709 V=800.0 PL=0
MOVL C00710 V=800.0 PL=0
MOVL C00711 V=800.0 PL=0
MOVL C00712 V=800.0 PL=0
MOVL C00713 V=800.0 PL=0
MOVL C00714 V=800.0 PL=0
MOVL C00715 V=800.0 PL=0
MOVL C00716 V=800.0 PL=0
MOVL C00717 V=800.0 PL=0
MOVL C00718 V=800.0 PL=0
MOVL C00719 V=800.0 PL=0
MOVL C00720 V=800.0 PL=0
MOVL C00721 V=800.0 PL=0
MOVL C00722 V=800.0 PL=0
MOVL C00723 V=800.0 PL=0
MOVL C00724 V=800.0 PL=0
MOVL C00725 V=800.0 PL=0
MOVL C00726 V=800.0 PL=0
MOVL C00727 V=800.0 PL=0
MOVL C00728 V=800.0 PL=0
MOVL C00729 V=800.0 PL=0
MOVL C00730 V=800.0 PL=0
MOVL C00731 V=800.0 PL=0
MOVL C00732 V=800.0 PL=0
MOVL C00733 V=800.0 PL=0
MOVL C00734 V=800.0 PL=0
MOVL C00735 V=800.0 PL=0
MOVL C00736 V=800.0 PL=0
MOVL C00737 V=800.0 PL=0
MOVL C00738 V=800.0 PL=0
MOVL C00739 V=800.0 PL=0
MOVL C00740 V=800.0 PL=0
MOVL C00741 V=800.0 PL=0
MOVL C00742 V=800.0 PL=0
MOVL C00743 V=800.0 PL=0
MOVL C00744 V=800.0 PL=0
MOVL C00745 V=800.0 PL=0
MOVL C00746 V=800.0 PL=0
MOVL C00747 V=800.0 PL=0
MOVL C00748 V=800.0 PL=0
MOVL C00749 V=800.0 PL=0
MOVL C00750 V=800.0 PL=0
MOVL C00751 V=800.0 PL=0
MOVL C00752 V=800.0 PL=0
MOVL C00753 V=800.0 PL=0
MOVL C00754 V=800.0 PL=0
MOVL C00755 V=800.0 PL=0
MOVL C00756 V=800.0 PL=0
MOVL C00757 V=800.0 PL=0
MOVL C00758 V=800.0 PL=0
MOVL C00759 V=800.0 PL=0
MOVL C00760 V=800.0 PL=0
MOVL C00761 V=800.0 PL=0
MOVL C00762 V=800.0 PL=0
MOVL C00763 V=800.0 PL=0
MOVL C00764 V=800.0 PL=0
MOVL C00765 V=800.0 PL=0
MOVL C00766 V=800.0 PL=0
MOVL C00767 V=800.0 PL=0
MOVL C00768 V=800.0 PL=0
MOVL C00769 V=800.0 PL=0
MOVL C00770 V=800.0 PL=0
MOVL C00771 V=800.0 PL=0
MOVL C00772 V=800.0 PL=0
MOVL C00773 V=800.0 PL=0
MOVL C00774 V=800.0 PL=0
MOVL C00775 V=800.0 PL=0
MOVL C00776 V=800.0 PL=0
MOVL C00777 V=800.0 PL=0
MOVL C00778 V=800.0 PL=0
MOVL C00779 V=800.0 PL=0
MOVL C00780 V=800.0 PL=0
MOVL C00781 V=800.0 PL=0
MOVL C00782 V=800.0 PL=0
MOVL C00783 V=800.0 PL=0
MOVL C00784 V=800.0 PL=0
MOVL C00785 V=800.0 PL=0
MOVL C00786 V=800.0 PL=0
MOVL C00787 V=800.0 PL=0
MOVL C00788 V=800.0 PL=0
MOVL C00789 V=800.0 PL=0
MOVL C00790 V=800.0 PL=0
MOVL C00791 V=800.0 PL=0
MOVL C00792 V=800.0 PL=0
MOVL C00793 V=800.0 PL=0
MOVL C00794 V=800.0 PL=0
MOVL C00795 V=800.0 PL=0
MOVL C00796 V=800.0 PL=0
MOVL C00797 V=800.0 PL=0
MOVL C00798 V=800.0 PL=0
MOVL C00799 V=800.0 PL=0
MOVL C00800 V=800.0 PL=0
MOVL C00801 V=800.0 PL=0
MOVL C00802 V=800.0 PL=0
MOVL C00803 V=800.0 PL=0
MOVL C00804 V=800.0 PL=0
MOVL C00805 V=800.0 PL=0
MOVL C00806 V=800.0 PL=0
MOVL C00807 V=800.0 PL=0
MOVL C00808 V=800.0 PL=0
MOVL C00809 V=800.0 PL=0
MOVL C00810 V=800.0 PL=0
MOVL C00811 V=800.0 PL=0
MOVL C00812 V=800.0 PL=0
MOVL C00813 V=800.0 PL=0
MOVL C00814 V=800.0 PL=0
MOVL C00815 V=800.0 PL=0
MOVL C00816 V=800.0 PL=0
MOVL C00817 V=800.0 PL=0
MOVL C00818 V=800.0 PL=0
MOVL C00819 V=800.0 PL=0
MOVL C00820 V=800.0 PL=0
MOVL C00821 V=800.0 PL=0
MOVL C00822 V=800.0 PL=0
MOVL C00823 V=800.0 PL=0
MOVL C00824 V=800.0 PL=0
MOVL C00825 V=800.0 PL=0
MOVL C00826 V=800.0 PL=0
MOVL C00827 V=800.0 PL=0
MOVL C00828 V=800.0 PL=0
MOVL C00829 V=800.0 PL=0
MOVL C00830 V=800.0 PL=0
MOVL C00831 V=800.0 PL=0
MOVL C00832 V=800.0 PL=0
MOVL C00833 V=800.0 PL=0
MOVL C00834 V=800.0 PL=0
MOVL C00835 V=800.0 PL=0
MOVL C00836 V=800.0 PL=0
MOVL C00837 V=800.0 PL=0
MOVL C00838 V=800.0 PL=0
MOVL C00839 V=800.0 PL=0
MOVL C00840 V=800.0 PL=0
MOVL C00841 V=800.0 PL=0
MOVL C00842 V=800.0 PL=0
MOVL C00843 V=800.0 PL=0
MOVL C00844 V=800.0 PL=0
MOVL C00845 V=800.0 PL=0
MOVL C00846 V=800.0 PL=0
MOVL C00847 V=800.0 PL=0
MOVL C00848 V=800.0 PL=0
MOVL C00849 V=800.0 PL=0
MOVL C00850 V=800.0 PL=0
MOVL C00851 V=800.0 PL=0
MOVL C00852 V=800.0 PL=0
MOVL C00853 V=800.0 PL=0
MOVL C00854 V=800.0 PL=0
MOVL C00855 V=800.0 PL=0
MOVL C00856 V=800.0 PL=0
MOVL C00857 V=800.0 PL=0
MOVL C00858 V=800.0 PL=0
MOVL C00859 V=800.0 PL=0
MOVL C00860 V=800.0 PL=0
MOVL C00861 V=800.0 PL=0
MOVL C00862 V=800.0 PL=0
MOVL C00863 V=800.0 PL=0
MOVL C00864 V=800.0 PL=0
MOVL C00865 V=800.0 PL=0
MOVL C00866 V=800.0 PL=0
MOVL C00867 V=800.0 PL=0
MOVL C00868 V=800.0 PL=0
MOVL C00869 V=800.0 PL=0
MOVL C00870 V=800.0 PL=0
MOVL C00871 V=800.0 PL=0
MOVL C00872 V=800.0 PL=0
MOVL C00873 V=800.0 PL=0
MOVL C00874 V=800.0 PL=0
MOVL C00875 V=800.0 PL=0
MOVL C00876 V=800.0 PL=0
MOVL C00877 V=800.0 PL=0
MOVL C00878 V=800.0 PL=0
MOVL C00879 V=800.0 PL=0
MOVL C00880 V=800.0 PL=0
MOVL C00881 V=800.0 PL=0
MOVL C00882 V=800.0 PL=0
MOVL C00883 V=800.0 PL=0
MOVL C00884 V=800.0 PL=0
MOVL C00885 V=800.0 PL=0
MOVL C00886 V=800.0 PL=0
MOVL C00887 V=800.0 PL=0
MOVL C00888 V=800.0 PL=0
MOVL C00889 V=800.0 PL=0
MOVL C00890 V=800.0 PL=0
MOVL C00891 V=800.0 PL=0
MOVL C00892 V=800.0 PL=0
MOVL C00893 V=800.0 PL=0
MOVL C00894 V=800.0 PL=0
MOVL C00895 V=800.0 PL=0
MOVL C00896 V=800.0 PL=0
MOVL C00897 V=800.0 PL=0
MOVL C00898 V=800.0 PL=0
MOVL C00899 V=800.0 PL=0
MOVL C00900 V=800.0 PL=0
MOVL C00901 V=800.0 PL=0
MOVL C00902 V=800.0 PL=0
MOVL C00903 V=800.0 PL=0
MOVL C00904 V=800.0 PL=0
MOVL C00905 V=800.0 PL=0
MOVL C00906 V=800.0 PL=0
MOVL C00907 V=800.0 PL=0
MOVL C00908 V=800.0 PL=0
MOVL C00909 V=800.0 PL=0
MOVL C00910 V=800.0 PL=0
MOVL C00911 V=800.0 PL=0
MOVL C00912 V=800.0 PL=0
MOVL C00913 V=800.0 PL=0
MOVL C00914 V=800.0 PL=0
MOVL C00915 V=800.0 PL=0
MOVL C00916 V=800.0 PL=0
MOVL C00917 V=800.0 PL=0
MOVL C00918 V=800.0 PL=0
MOVL C00919 V=800.0 PL=0
MOVL C00920 V=800.0 PL=0
MOVL C00921 V=800.0 PL=0
MOVL C00922 V=800.0 PL=0
MOVL C00923 V=800.0 PL=0
MOVL C00924 V=800.0 PL=0
MOVL C00925 V=800.0 PL=0
MOVL C00926 V=800.0 PL=0
MOVL C00927 V=800.0 PL=0
MOVL C00928 V=800.0 PL=0
MOVL C00929 V=800.0 PL=0
MOVL C00930 V=800.0 PL=0
MOVL C00931 V=800.0 PL=0
MOVL C00932 V=800.0 PL=0
MOVL C00933 V=800.0 PL=0
MOVL C00934 V=800.0 PL=0
MOVL C00935 V=800.0 PL=0
MOVL C00936 V=800.0 PL=0
MOVL C00937 V=800.0 PL=0
MOVL C00938 V=800.0 PL=0
MOVL C00939 V=800.0 PL=0
MOVL C00940 V=800.0 PL=0
MOVL C00941 V=800.0 PL=0
MOVL C00942 V=800.0 PL=0
MOVL C00943 V=800.0 PL=0
MOVL C00944 V=800.0 PL=0
MOVL C00945 V=800.0 PL=0
MOVL C00946 V=800.0 PL=0
MOVL C00947 V=800.0 PL=0
MOVL C00948 V=800.0 PL=0
MOVL C00949 V=800.0 PL=0
MOVL C00950 V=800.0 PL=0
MOVL C00951 V=800.0 PL=0
MOVL C00952 V=800.0 PL=0
MOVL C00953 V=800.0 PL=0
MOVL C00954 V=800.0 PL=0
MOVL C00955 V=800.0 PL=0
MOVL C00956 V=800.0 PL=0
MOVL C00957 V=800.0 PL=0
MOVL C00958 V=800.0 PL=0
MOVL C00959 V=800.0 PL=0
MOVL C00960 V=800.0 PL=0
MOVL C00961 V=800.0 PL=0
MOVL C00962 V=800.0 PL=0
MOVL C00963 V=800.0 PL=0
MOVL C00964 V=800.0 PL=0
MOVL C00965 V=800.0 PL=0
MOVL C00966 V=800.0 PL=0
MOVL C00967 V=800.0 PL=0
MOVL C00968 V=800.0 PL=0
MOVL C00969 V=800.0 PL=0
MOVL C00970 V=800.0 PL=0
MOVL C00971 V=800.0 PL=0
MOVL C00972 V=800.0 PL=0
MOVL C00973 V=800.0 PL=0
MOVL C00974 V=800.0 PL=0
MOVL C00975 V=800.0 PL=0
MOVL C00976 V=800.0 PL=0
MOVL C00977 V=800.0 PL=0
MOVL C00978 V=800.0 PL=0
MOVL C00979 V=800.0 PL=0
MOVL C00980 V=800.0 PL=0
MOVL C00981 V=800.0 PL=0
MOVL C00982 V=800.0 PL=0
MOVL C00983 V=800.0 PL=0
MOVL C00984 V=800.0 PL=0
MOVL C00985 V=800.0 PL=0
MOVL C00986 V=800.0 PL=0
MOVL C00987 V=800.0 PL=0
MOVL C00988 V=800.0 PL=0
MOVL C00989 V=800.0 PL=0
MOVL C00990 V=800.0 PL=0
MOVL C00991 V=800.0 PL=0
MOVL C00992 V=800.0 PL=0
MOVL C00993 V=800.0 PL=0
MOVL C00994 V=800.0 PL=0
MOVL C00995 V=800.0 PL=0
MOVL C00996 V=800.0 PL=0
MOVL C00997 V=800.0 PL=0
MOVL C00998 V=800.0 PL=0
MOVL C00999 V=800.0 PL=0
MOVL C01000 V=800.0 PL=0
MOVL C01001 V=800.0 PL=0
MOVL C01002 V=800.0 PL=0
MOVL C01003 V=800.0 PL=0
MOVL C01004 V=800.0 PL=0
MOVL C01005 V=800.0 PL=0
MOVL C01006 V=800.0 PL=0
MOVL C01007 V=800.0 PL=0
MOVL C01008 V=800.0 PL=0
MOVL C01009 V=800.0 PL=0
MOVL C01010 V=800.0 PL=0
MOVL C01011 V=800.0 PL=0
MOVL C01012 V=800.0 PL=0
MOVL C01013 V=800.0 PL=0
MOVL C01014 V=800.0 PL=0
MOVL C01015 V=800.0 PL=0
MOVL C01016 V=800.0 PL=0
MOVL C01017 V=800.0 PL=0
MOVL C01018 V=800.0 PL=0
MOVL C01019 V=800.0 PL=0
MOVL C01020 V=800.0 PL=0
MOVL C01021 V=800.0 PL=0
MOVL C01022 V=800.0 PL=0
MOVL C01023 V=800.0 PL=0
MOVL C01024 V=800.0 PL=0
MOVL C01025 V=800.0 PL=0
MOVL C01026 V=800.0 PL=0
MOVL C01027 V=800.0 PL=0
MOVL C01028 V=800.0 PL=0
MOVL C01029 V=800.0 PL=0
MOVL C01030 V=800.0 PL=0
MOVL C01031 V=800.0 PL=0
MOVL C01032 V=800.0 PL=0
MOVL C01033 V=800.0 PL=0
MOVL C01034 V=800.0 PL=0
MOVL C01035 V=800.0 PL=0
MOVL C01036 V=800.0 PL=0
MOVL C01037 V=800.0 PL=0
MOVL C01038 V=800.0 PL=0
MOVL C01039 V=800.0 PL=0
MOVL C01040 V=800.0 PL=0
MOVL C01041 V=800.0 PL=0
MOVL C01042 V=800.0 PL=0
MOVL C01043 V=800.0 PL=0
MOVL C01044 V=800.0 PL=0
MOVL C01045 V=800.0 PL=0
MOVL C01046 V=800.0 PL=0
MOVL C01047 V=800.0 PL=0
MOVL C01048 V=800.0 PL=0
MOVL C01049 V=800.0 PL=0
MOVL C01050 V=800.0 PL=0
MOVL C01051 V=800.0 PL=0
MOVL C01052 V=800.0 PL=0
MOVL C01053 V=800.0 PL=0
MOVL C01054 V=800.0 PL=0
MOVL C01055 V=800.0 PL=0
MOVL C01056 V=800.0 PL=0
MOVL C01057 V=800.0 PL=0
MOVL C01058 V=800.0 PL=0
MOVL C01059 V=800.0 PL=0
MOVL C01060 V=800.0 PL=0
MOVL C01061 V=800.0 PL=0
MOVL C01062 V=800.0 PL=0
MOVL C01063 V=800.0 PL=0
MOVL C01064 V=800.0 PL=0
MOVL C01065 V=800.0 PL=0
MOVL C01066 V=800.0 PL=0
MOVL C01067 V=800.0 PL=0
MOVL C01068 V=800.0 PL=0
MOVL C01069 V=800.0 PL=0
MOVL C01070 V=800.0 PL=0
MOVL C01071 V=800.0 PL=0
MOVL C01072 V=800.0 PL=0
MOVL C01073 V=800.0 PL=0
MOVL C01074 V=800.0 PL=0
MOVL C01075 V=800.0 PL=0
MOVL C01076 V=800.0 PL=0
MOVL C01077 V=800.0 PL=0
MOVL C01078 V=800.0 PL=0
MOVL C01079 V=800.0 PL=0
MOVL C01080 V=800.0 PL=0
MOVL C01081 V=800.0 PL=0
MOVL C01082 V=800.0 PL=0
MOVL C01083 V=800.0 PL=0
MOVL C01084 V=800.0 PL=0
MOVL C01085 V=800.0 PL=0
MOVL C01086 V=800.0 PL=0
MOVL C01087 V=800.0 PL=0
MOVL C01088 V=800.0 PL=0
MOVL C01089 V=800.0 PL=0
MOVL C01090 V=800.0 PL=0
MOVL C01091 V=800.0 PL=0
MOVL C01092 V=800.0 PL=0
MOVL C01093 V=800.0 PL=0
MOVL C01094 V=800.0 PL=0
MOVL C01095 V=800.0 PL=0
MOVL C01096 V=800.0 PL=0
MOVL C01097 V=800.0 PL=0
MOVL C01098 V=800.0 PL=0
MOVL C01099 V=800.0 PL=0
MOVL C01100 V=800.0 PL=0
MOVL C01101 V=800.0 PL=0
MOVL C01102 V=800.0 PL=0
MOVL C01103 V=800.0 PL=0
MOVL C01104 V=800.0 PL=0
MOVL C01105 V=800.0 PL=0
MOVL C01106 V=800.0 PL=0
MOVL C01107 V=800.0 PL=0
MOVL C01108 V=800.0 PL=0
MOVL C01109 V=800.0 PL=0
MOVL C01110 V=800.0 PL=0
MOVL C01111 V=800.0 PL=0
MOVL C01112 V=800.0 PL=0
MOVL C01113 V=800.0 PL=0
MOVL C01114 V=800.0 PL=0
MOVL C01115 V=800.0 PL=0
MOVL C01116 V=800.0 PL=0
MOVL C01117 V=800.0 PL=0
MOVL C01118 V=800.0 PL=0
MOVL C01119 V=800.0 PL=0
MOVL C01120 V=800.0 PL=0
MOVL C01121 V=800.0 PL=0
MOVL C01122 V=800.0 PL=0
MOVL C01123 V=800.0 PL=0
MOVL C01124 V=800.0 PL=0
MOVL C01125 V=800.0 PL=0
MOVL C01126 V=800.0 PL=0
MOVL C01127 V=800.0 PL=0
MOVL C01128 V=800.0 PL=0
MOVL C01129 V=800.0 PL=0
MOVL C01130 V=800.0 PL=0
MOVL C01131 V=800.0 PL=0
MOVL C01132 V=800.0 PL=0
MOVL C01133 V=800.0 PL=0
MOVL C01134 V=800.0 PL=0
MOVL C01135 V=800.0 PL=0
MOVL C01136 V=800.0 PL=0
MOVL C01137 V=800.0 PL=0
MOVL C01138 V=800.0 PL=0
MOVL C01139 V=800.0 PL=0
MOVL C01140 V=800.0 PL=0
MOVL C01141 V=800.0 PL=0
MOVL C01142 V=800.0 PL=0
MOVL C01143 V=800.0 PL=0
MOVL C01144 V=800.0 PL=0
MOVL C01145 V=800.0 PL=0
MOVL C01146 V=800.0 PL=0
MOVL C01147 V=800.0 PL=0
MOVL C01148 V=800.0 PL=0
MOVL C01149 V=800.0 PL=0
MOVL C01150 V=800.0 PL=0
MOVL C01151 V=800.0 PL=0
MOVL C01152 V=800.0 PL=0
MOVL C01153 V=800.0 PL=0
MOVL C01154 V=800.0 PL=0
MOVL C01155 V=800.0 PL=0
MOVL C01156 V=800.0 PL=0
MOVL C01157 V=800.0 PL=0
MOVL C01158 V=800.0 PL=0
MOVL C01159 V=800.0 PL=0
MOVL C01160 V=800.0 PL=0
MOVL C01161 V=800.0 PL=0
MOVL C01162 V=800.0 PL=0
MOVL C01163 V=800.0 PL=0
MOVL C01164 V=800.0 PL=0
MOVL C01165 V=800.0 PL=0
MOVL C01166 V=800.0 PL=0
MOVL C01167 V=800.0 PL=0
MOVL C01168 V=800.0 PL=0
MOVL C01169 V=800.0 PL=0
MOVL C01170 V=800.0 PL=0
MOVL C01171 V=800.0 PL=0
MOVL C01172 V=800.0 PL=0
MOVL C01173 V=800.0 PL=0
MOVL C01174 V=800.0 PL=0
MOVL C01175 V=800.0 PL=0
MOVL C01176 V=800.0 PL=0
MOVL C01177 V=800.0 PL=0
MOVL C01178 V=800.0 PL=0
MOVL C01179 V=800.0 PL=0
MOVL C01180 V=800.0 PL=0
MOVL C01181 V=800.0 PL=0
MOVL C01182 V=800.0 PL=0
MOVL C01183 V=800.0 PL=0
MOVL C01184 V=800.0 PL=0
MOVL C01185 V=800.0 PL=0
MOVL C01186 V=800.0 PL=0
MOVL C01187 V=800.0 PL=0
MOVL C01188 V=800.0 PL=0
MOVL C01189 V=800.0 PL=0
MOVL C01190 V=800.0 PL=0
MOVL C01191 V=800.0 PL=0
MOVL C01192 V=800.0 PL=0
MOVL C01193 V=800.0 PL=0
MOVL C01194 V=800.0 PL=0
MOVL C01195 V=800.0 PL=0
MOVL C01196 V=800.0 PL=0
MOVL C01197 V=800.0 PL=0
MOVL C01198 V=800.0 PL=0
MOVL C01199 V=800.0 PL=0
MOVL C01200 V=800.0 PL=0
MOVL C01201 V=800.0 PL=0
MOVL C01202 V=800.0 PL=0
MOVL C01203 V=800.0 PL=0
MOVL C01204 V=800.0 PL=0
MOVL C01205 V=800.0 PL=0
MOVL C01206 V=800.0 PL=0
MOVL C01207 V=800.0 PL=0
MOVL C01208 V=800.0 PL=0
MOVL C01209 V=800.0 PL=0
MOVL C01210 V=800.0 PL=0
MOVL C01211 V=800.0 PL=0
MOVL C01212 V=800.0 PL=0
MOVL C01213 V=800.0 PL=0
MOVL C01214 V=800.0 PL=0
MOVL C01215 V=800.0 PL=0
MOVL C01216 V=800.0 PL=0
MOVL C01217 V=800.0 PL=0
MOVL C01218 V=800.0 PL=0
MOVL C01219 V=800.0 PL=0
MOVL C01220 V=800.0 PL=0
MOVL C01221 V=800.0 PL=0
MOVL C01222 V=800.0 PL=0
MOVL C01223 V=800.0 PL=0
MOVL C01224 V=800.0 PL=0
MOVL C01225 V=800.0 PL=0
MOVL C01226 V=800.0 PL=0
MOVL C01227 V=800.0 PL=0
MOVL C01228 V=800.0 PL=0
MOVL C01229 V=800.0 PL=0
MOVL C01230 V=800.0 PL=0
MOVL C01231 V=800.0 PL=0
MOVL C01232 V=800.0 PL=0
MOVL C01233 V=800.0 PL=0
MOVL C01234 V=800.0 PL=0
MOVL C01235 V=800.0 PL=0
MOVL C01236 V=800.0 PL=0
MOVL C01237 V=800.0 PL=0
MOVL C01238 V=800.0 PL=0
MOVL C01239 V=800.0 PL=0
MOVL C01240 V=800.0 PL=0
MOVL C01241 V=800.0 PL=0
MOVL C01242 V=800.0 PL=0
MOVL C01243 V=800.0 PL=0
MOVL C01244 V=800.0 PL=0
MOVL C01245 V=800.0 PL=0
MOVL C01246 V=800.0 PL=0
MOVL C01247 V=800.0 PL=0
MOVL C01248 V=800.0 PL=0
MOVL C01249 V=800.0 PL=0
MOVL C01250 V=800.0 PL=0
MOVL C01251 V=800.0 PL=0
MOVL C01252 V=800.0 PL=0
MOVL C01253 V=800.0 PL=0
MOVL C01254 V=800.0 PL=0
MOVL C01255 V=800.0 PL=0
MOVL C01256 V=800.0 PL=0
MOVL C01257 V=800.0 PL=0
MOVL C01258 V=800.0 PL=0
MOVL C01259 V=800.0 PL=0
MOVL C01260 V=800.0 PL=0
MOVL C01261 V=800.0 PL=0
MOVL C01262 V=800.0 PL=0
MOVL C01263 V=800.0 PL=0
MOVL C01264 V=800.0 PL=0
MOVL C01265 V=800.0 PL=0
MOVL C01266 V=800.0 PL=0
MOVL C01267 V=800.0 PL=0
MOVL C01268 V=800.0 PL=0
MOVL C01269 V=800.0 PL=0
MOVL C01270 V=800.0 PL=0
MOVL C01271 V=800.0 PL=0
MOVL C01272 V=800.0 PL=0
MOVL C01273 V=800.0 PL=0
MOVL C01274 V=800.0 PL=0
MOVL C01275 V=800.0 PL=0
MOVL C01276 V=800.0 PL=0
MOVL C01277 V=800.0 PL=0
MOVL C01278 V=800.0 PL=0
MOVL C01279 V=800.0 PL=0
MOVL C01280 V=800.0 PL=0
MOVL C01281 V=800.0 PL=0
MOVL C01282 V=800.0 PL=0
MOVL C01283 V=800.0 PL=0
MOVL C01284 V=800.0 PL=0
MOVL C01285 V=800.0 PL=0
MOVL C01286 V=800.0 PL=0
MOVL C01287 V=800.0 PL=0
MOVL C01288 V=800.0 PL=0
MOVL C01289 V=800.0 PL=0
MOVL C01290 V=800.0 PL=0
MOVL C01291 V=800.0 PL=0
MOVL C01292 V=800.0 PL=0
MOVL C01293 V=800.0 PL=0
MOVL C01294 V=800.0 PL=0
MOVL C01295 V=800.0 PL=0
MOVL C01296 V=800.0 PL=0
MOVL C01297 V=800.0 PL=0
MOVL C01298 V=800.0 PL=0
MOVL C01299 V=800.0 PL=0
MOVL C01300 V=800.0 PL=0
MOVL C01301 V=800.0 PL=0
MOVL C01302 V=800.0 PL=0
MOVL C01303 V=800.0 PL=0
MOVL C01304 V=800.0 PL=0
MOVL C01305 V=800.0 PL=0
MOVL C01306 V=800.0 PL=0
MOVL C01307 V=800.0 PL=0
MOVL C01308 V=800.0 PL=0
MOVL C01309 V=800.0 PL=0
MOVL C01310 V=800.0 PL=0
MOVL C01311 V=800.0 PL=0
MOVL C01312 V=800.0 PL=0
MOVL C01313 V=800.0 PL=0
MOVL C01314 V=800.0 PL=0
MOVL C01315 V=800.0 PL=0
MOVL C01316 V=800.0 PL=0
MOVL C01317 V=800.0 PL=0
MOVL C01318 V=800.0 PL=0
MOVL C01319 V=800.0 PL=0
MOVL C01320 V=800.0 PL=0
MOVL C01321 V=800.0 PL=0
MOVL C01322 V=800.0 PL=0
MOVL C01323 V=800.0 PL=0
MOVL C01324 V=800.0 PL=0
MOVL C01325 V=800.0 PL=0
MOVL C01326 V=800.0 PL=0
MOVL C01327 V=800.0 PL=0
MOVL C01328 V=800.0 PL=0
MOVL C01329 V=800.0 PL=0
MOVL C01330 V=800.0 PL=0
MOVL C01331 V=800.0 PL=0
MOVL C01332 V=800.0 PL=0
MOVL C01333 V=800.0 PL=0
MOVL C01334 V=800.0 PL=0
MOVL C01335 V=800.0 PL=0
MOVL C01336 V=800.0 PL=0
MOVL C01337 V=800.0 PL=0
MOVL C01338 V=800.0 PL=0
MOVL C01339 V=800.0 PL=0
MOVL C01340 V=800.0 PL=0
MOVL C01341 V=800.0 PL=0
MOVL C01342 V=800.0 PL=0
MOVL C01343 V=800.0 PL=0
MOVL C01344 V=800.0 PL=0
MOVL C01345 V=800.0 PL=0
MOVL C01346 V=800.0 PL=0
MOVL C01347 V=800.0 PL=0
MOVL C01348 V=800.0 PL=0
MOVL C01349 V=800.0 PL=0
MOVL C01350 V=800.0 PL=0
MOVL C01351 V=800.0 PL=0
MOVL C01352 V=800.0 PL=0
MOVL C01353 V=800.0 PL=0
MOVL C01354 V=800.0 PL=0
MOVL C01355 V=800.0 PL=0
MOVL C01356 V=800.0 PL=0
MOVL C01357 V=800.0 PL=0
MOVL C01358 V=800.0 PL=0
MOVL C01359 V=800.0 PL=0
MOVL C01360 V=800.0 PL=0
MOVL C01361 V=800.0 PL=0
MOVL C01362 V=800.0 PL=0
MOVL C01363 V=800.0 PL=0
MOVL C01364 V=800.0 PL=0
MOVL C01365 V=800.0 PL=0
MOVL C01366 V=800.0 PL=0
MOVL C01367 V=800.0 PL=0
MOVL C01368 V=800.0 PL=0
MOVL C01369 V=800.0 PL=0
MOVL C01370 V=800.0 PL=0
MOVL C01371 V=800.0 PL=0
MOVL C01372 V=800.0 PL=0
MOVL C01373 V=800.0 PL=0
MOVL C01374 V=800.0 PL=0
MOVL C01375 V=800.0 PL=0
MOVL C01376 V=800.0 PL=0
MOVL C01377 V=800.0 PL=0
MOVL C01378 V=800.0 PL=0
MOVL C01379 V=800.0 PL=0
MOVL C01380 V=800.0 PL=0
MOVL C01381 V=800.0 PL=0
MOVL C01382 V=800.0 PL=0
MOVL C01383 V=800.0 PL=0
MOVL C01384 V=800.0 PL=0
MOVL C01385 V=800.0 PL=0
MOVL C01386 V=800.0 PL=0
MOVL C01387 V=800.0 PL=0
MOVL C01388 V=800.0 PL=0
MOVL C01389 V=800.0 PL=0
MOVL C01390 V=800.0 PL=0
MOVL C01391 V=800.0 PL=0
MOVL C01392 V=800.0 PL=0
MOVL C01393 V=800.0 PL=0
MOVL C01394 V=800.0 PL=0
MOVL C01395 V=800.0 PL=0
MOVL C01396 V=800.0 PL=0
MOVL C01397 V=800.0 PL=0
MOVL C01398 V=800.0 PL=0
MOVL C01399 V=800.0 PL=0
MOVL C01400 V=800.0 PL=0
MOVL C01401 V=800.0 PL=0
MOVL C01402 V=800.0 PL=0
MOVL C01403 V=800.0 PL=0
MOVL C01404 V=800.0 PL=0
MOVL C01405 V=800.0 PL=0
MOVL C01406 V=800.0 PL=0
MOVL C01407 V=800.0 PL=0
MOVL C01408 V=800.0 PL=0
MOVL C01409 V=800.0 PL=0
MOVL C01410 V=800.0 PL=0
MOVL C01411 V=800.0 PL=0
MOVL C01412 V=800.0 PL=0
MOVL C01413 V=800.0 PL=0
MOVL C01414 V=800.0 PL=0
MOVL C01415 V=800.0 PL=0
MOVL C01416 V=800.0 PL=0
MOVL C01417 V=800.0 PL=0
MOVL C01418 V=800.0 PL=0
MOVL C01419 V=800.0 PL=0
MOVL C01420 V=800.0 PL=0
MOVL C01421 V=800.0 PL=0
MOVL C01422 V=800.0 PL=0
MOVL C01423 V=800.0 PL=0
MOVL C01424 V=800.0 PL=0
MOVL C01425 V=800.0 PL=0
MOVL C01426 V=800.0 PL=0
MOVL C01427 V=800.0 PL=0
MOVL C01428 V=800.0 PL=0
MOVL C01429 V=800.0 PL=0
MOVL C01430 V=800.0 PL=0
MOVL C01431 V=800.0 PL=0
MOVL C01432 V=800.0 PL=0
MOVL C01433 V=800.0 PL=0
MOVL C01434 V=800.0 PL=0
MOVL C01435 V=800.0 PL=0
MOVL C01436 V=800.0 PL=0
MOVL C01437 V=800.0 PL=0
MOVL C01438 V=800.0 PL=0
MOVL C01439 V=800.0 PL=0
MOVL C01440 V=800.0 PL=0
MOVL C01441 V=800.0 PL=0
MOVL C01442 V=800.0 PL=0
MOVL C01443 V=800.0 PL=0
MOVL C01444 V=800.0 PL=0
MOVL C01445 V=800.0 PL=0
MOVL C01446 V=800.0 PL=0
MOVL C01447 V=800.0 PL=0
MOVL C01448 V=800.0 PL=0
MOVL C01449 V=800.0 PL=0
MOVL C01450 V=800.0 PL=0
MOVL C01451 V=800.0 PL=0
MOVL C01452 V=800.0 PL=0
MOVL C01453 V=800.0 PL=0
MOVL C01454 V=800.0 PL=0
MOVL C01455 V=800.0 PL=0
MOVL C01456 V=800.0 PL=0
MOVL C01457 V=800.0 PL=0
MOVL C01458 V=800.0 PL=0
MOVL C01459 V=800.0 PL=0
MOVL C01460 V=800.0 PL=0
MOVL C01461 V=800.0 PL=0
MOVL C01462 V=800.0 PL=0
MOVL C01463 V=800.0 PL=0
MOVL C01464 V=800.0 PL=0
MOVL C01465 V=800.0 PL=0
MOVL C01466 V=800.0 PL=0
MOVL C01467 V=800.0 PL=0
MOVL C01468 V=800.0 PL=0
MOVL C01469 V=800.0 PL=0
MOVL C01470 V=800.0 PL=0
MOVL C01471 V=800.0 PL=0
MOVL C01472 V=800.0 PL=0
MOVL C01473 V=800.0 PL=0
MOVL C01474 V=800.0 PL=0
MOVL C01475 V=800.0 PL=0
MOVL C01476 V=800.0 PL=0
MOVL C01477 V=800.0 PL=0
MOVL C01478 V=800.0 PL=0
MOVL C01479 V=800.0 PL=0
MOVL C01480 V=800.0 PL=0
MOVL C01481 V=800.0 PL=0
MOVL C01482 V=800.0 PL=0
MOVL C01483 V=800.0 PL=0
MOVL C01484 V=800.0 PL=0
MOVL C01485 V=800.0 PL=0
MOVL C01486 V=800.0 PL=0
MOVL C01487 V=800.0 PL=0
MOVL C01488 V=800.0 PL=0
MOVL C01489 V=800.0 PL=0
MOVL C01490 V=800.0 PL=0
MOVL C01491 V=800.0 PL=0
MOVL C01492 V=800.0 PL=0
MOVL C01493 V=800.0 PL=0
MOVL C01494 V=800.0 PL=0
MOVL C01495 V=800.0 PL=0
MOVL C01496 V=800.0 PL=0
MOVL C01497 V=800.0 PL=0
MOVL C01498 V=800.0 PL=0
MOVL C01499 V=800.0 PL=0
MOVL C01500 V=800.0 PL=0
MOVL C01501 V=800.0 PL=0
MOVL C01502 V=800.0 PL=0
MOVL C01503 V=800.0 PL=0
MOVL C01504 V=800.0 PL=0
MOVL C01505 V=800.0 PL=0
MOVL C01506 V=800.0 PL=0
MOVL C01507 V=800.0 PL=0
MOVL C01508 V=800.0 PL=0
MOVL C01509 V=800.0 PL=0
MOVL C01510 V=800.0 PL=0
MOVL C01511 V=800.0 PL=0
MOVL C01512 V=800.0 PL=0
MOVL C01513 V=800.0 PL=0
MOVL C01514 V=800.0 PL=0
MOVL C01515 V=800.0 PL=0
MOVL C01516 V=800.0 PL=0
MOVL C01517 V=800.0 PL=0
MOVL C01518 V=800.0 PL=0
MOVL C01519 V=800.0 PL=0
MOVL C01520 V=800.0 PL=0
MOVL C01521 V=800.0 PL=0
MOVL C01522 V=800.0 PL=0
MOVL C01523 V=800.0 PL=0
MOVL C01524 V=800.0 PL=0
MOVL C01525 V=800.0 PL=0
MOVL C01526 V=800.0 PL=0
MOVL C01527 V=800.0 PL=0
MOVL C01528 V=800.0 PL=0
MOVL C01529 V=800.0 PL=0
MOVL C01530 V=800.0 PL=0
MOVL C01531 V=800.0 PL=0
MOVL C01532 V=800.0 PL=0
MOVL C01533 V=800.0 PL=0
MOVL C01534 V=800.0 PL=0
MOVL C01535 V=800.0 PL=0
MOVL C01536 V=800.0 PL=0
MOVL C01537 V=800.0 PL=0
MOVL C01538 V=800.0 PL=0
MOVL C01539 V=800.0 PL=0
MOVL C01540 V=800.0 PL=0
MOVL C01541 V=800.0 PL=0
MOVL C01542 V=800.0 PL=0
MOVL C01543 V=800.0 PL=0
MOVL C01544 V=800.0 PL=0
MOVL C01545 V=800.0 PL=0
MOVL C01546 V=800.0 PL=0
MOVL C01547 V=800.0 PL=0
MOVL C01548 V=800.0 PL=0
MOVL C01549 V=800.0 PL=0
MOVL C01550 V=800.0 PL=0
MOVL C01551 V=800.0 PL=0
MOVL C01552 V=800.0 PL=0
MOVL C01553 V=800.0 PL=0
MOVL C01554 V=800.0 PL=0
MOVL C01555 V=800.0 PL=0
MOVL C01556 V=800.0 PL=0
MOVL C01557 V=800.0 PL=0
MOVL C01558 V=800.0 PL=0
MOVL C01559 V=800.0 PL=0
MOVL C01560 V=800.0 PL=0
MOVL C01561 V=800.0 PL=0
MOVL C01562 V=800.0 PL=0
MOVL C01563 V=800.0 PL=0
MOVL C01564 V=800.0 PL=0
MOVL C01565 V=800.0 PL=0
MOVL C01566 V=800.0 PL=0
MOVL C01567 V=800.0 PL=0
MOVL C01568 V=800.0 PL=0
MOVL C01569 V=800.0 PL=0
MOVL C01570 V=800.0 PL=0
MOVL C01571 V=800.0 PL=0
MOVL C01572 V=800.0 PL=0
MOVL C01573 V=800.0 PL=0
MOVL C01574 V=800.0 PL=0
MOVL C01575 V=800.0 PL=0
MOVL C01576 V=800.0 PL=0
MOVL C01577 V=800.0 PL=0
MOVL C01578 V=800.0 PL=0
MOVL C01579 V=800.0 PL=0
MOVL C01580 V=800.0 PL=0
MOVL C01581 V=800.0 PL=0
MOVL C01582 V=800.0 PL=0
MOVL C01583 V=800.0 PL=0
MOVL C01584 V=800.0 PL=0
MOVL C01585 V=800.0 PL=0
MOVL C01586 V=800.0 PL=0
MOVL C01587 V=800.0 PL=0
MOVL C01588 V=800.0 PL=0
MOVL C01589 V=800.0 PL=0
MOVL C01590 V=800.0 PL=0
MOVL C01591 V=800.0 PL=0
MOVL C01592 V=800.0 PL=0
MOVL C01593 V=800.0 PL=0
MOVL C01594 V=800.0 PL=0
MOVL C01595 V=800.0 PL=0
MOVL C01596 V=800.0 PL=0
MOVL C01597 V=800.0 PL=0
MOVL C01598 V=800.0 PL=0
MOVL C01599 V=800.0 PL=0
MOVL C01600 V=800.0 PL=0
MOVL C01601 V=800.0 PL=0
MOVL C01602 V=800.0 PL=0
MOVL C01603 V=800.0 PL=0
MOVL C01604 V=800.0 PL=0
MOVL C01605 V=800.0 PL=0
MOVL C01606 V=800.0 PL=0
MOVL C01607 V=800.0 PL=0
MOVL C01608 V=800.0 PL=0
MOVL C01609 V=800.0 PL=0
MOVL C01610 V=800.0 PL=0
MOVL C01611 V=800.0 PL=0
MOVL C01612 V=800.0 PL=0
MOVL C01613 V=800.0 PL=0
MOVL C01614 V=800.0 PL=0
MOVL C01615 V=800.0 PL=0
MOVL C01616 V=800.0 PL=0
MOVL C01617 V=800.0 PL=0
MOVL C01618 V=800.0 PL=0
MOVL C01619 V=800.0 PL=0
MOVL C01620 V=800.0 PL=0
MOVL C01621 V=800.0 PL=0
MOVL C01622 V=800.0 PL=0
MOVL C01623 V=800.0 PL=0
MOVL C01624 V=800.0 PL=0
MOVL C01625 V=800.0 PL=0
MOVL C01626 V=800.0 PL=0
MOVL C01627 V=800.0 PL=0
MOVL C01628 V=800.0 PL=0
MOVL C01629 V=800.0 PL=0
MOVL C01630 V=800.0 PL=0
MOVL C01631 V=800.0 PL=0
MOVL C01632 V=800.0 PL=0
MOVL C01633 V=800.0 PL=0
MOVL C01634 V=800.0 PL=0
MOVL C01635 V=800.0 PL=0
MOVL C01636 V=800.0 PL=0
MOVL C01637 V=800.0 PL=0
MOVL C01638 V=800.0 PL=0
MOVL C01639 V=800.0 PL=0
MOVL C01640 V=800.0 PL=0
MOVL C01641 V=800.0 PL=0
MOVL C01642 V=800.0 PL=0
MOVL C01643 V=800.0 PL=0
MOVL C01644 V=800.0 PL=0
MOVL C01645 V=800.0 PL=0
MOVL C01646 V=800.0 PL=0
MOVL C01647 V=800.0 PL=0
MOVL C01648 V=800.0 PL=0
MOVL C01649 V=800.0 PL=0
MOVL C01650 V=800.0 PL=0
MOVL C01651 V=800.0 PL=0
MOVL C01652 V=800.0 PL=0
MOVL C01653 V=800.0 PL=0
MOVL C01654 V=800.0 PL=0
MOVL C01655 V=800.0 PL=0
MOVL C01656 V=800.0 PL=0
MOVL C01657 V=800.0 PL=0
MOVL C01658 V=800.0 PL=0
MOVL C01659 V=800.0 PL=0
MOVL C01660 V=800.0 PL=0
MOVL C01661 V=800.0 PL=0
MOVL C01662 V=800.0 PL=0
MOVL C01663 V=800.0 PL=0
MOVL C01664 V=800.0 PL=0
MOVL C01665 V=800.0 PL=0
MOVL C01666 V=800.0 PL=0
MOVL C01667 V=800.0 PL=0
MOVL C01668 V=800.0 PL=0
MOVL C01669 V=800.0 PL=0
MOVL C01670 V=800.0 PL=0
MOVL C01671 V=800.0 PL=0
MOVL C01672 V=800.0 PL=0
MOVL C01673 V=800.0 PL=0
MOVL C01674 V=800.0 PL=0
MOVL C01675 V=800.0 PL=0
MOVL C01676 V=800.0 PL=0
MOVL C01677 V=800.0 PL=0
MOVL C01678 V=800.0 PL=0
MOVL C01679 V=800.0 PL=0
MOVL C01680 V=800.0 PL=0
MOVL C01681 V=800.0 PL=0
MOVL C01682 V=800.0 PL=0
MOVL C01683 V=800.0 PL=0
MOVL C01684 V=800.0 PL=0
MOVL C01685 V=800.0 PL=0
MOVL C01686 V=800.0 PL=0
MOVL C01687 V=800.0 PL=0
MOVL C01688 V=800.0 PL=0
MOVL C01689 V=800.0 PL=0
MOVL C01690 V=800.0 PL=0
MOVL C01691 V=800.0 PL=0
MOVL C01692 V=800.0 PL=0
MOVL C01693 V=800.0 PL=0
MOVL C01694 V=800.0 PL=0
MOVL C01695 V=800.0 PL=0
MOVL C01696 V=800.0 PL=0
MOVL C01697 V=800.0 PL=0
MOVL C01698 V=800.0 PL=0
MOVL C01699 V=800.0 PL=0
MOVL C01700 V=800.0 PL=0
MOVL C01701 V=800.0 PL=0
MOVL C01702 V=800.0 PL=0
MOVL C01703 V=800.0 PL=0
MOVL C01704 V=800.0 PL=0
MOVL C01705 V=800.0 PL=0
MOVL C01706 V=800.0 PL=0
MOVL C01707 V=800.0 PL=0
MOVL C01708 V=800.0 PL=0
MOVL C01709 V=800.0 PL=0
MOVL C01710 V=800.0 PL=0
MOVL C01711 V=800.0 PL=0
MOVL C01712 V=800.0 PL=0
MOVL C01713 V=800.0 PL=0
MOVL C01714 V=800.0 PL=0
MOVL C01715 V=800.0 PL=0
MOVL C01716 V=800.0 PL=0
MOVL C01717 V=800.0 PL=0
MOVL C01718 V=800.0 PL=0
MOVL C01719 V=800.0 PL=0
MOVL C01720 V=800.0 PL=0
MOVL C01721 V=800.0 PL=0
MOVL C01722 V=800.0 PL=0
MOVL C01723 V=800.0 PL=0
MOVL C01724 V=800.0 PL=0
MOVL C01725 V=800.0 PL=0
MOVL C01726 V=800.0 PL=0
MOVL C01727 V=800.0 PL=0
MOVL C01728 V=800.0 PL=0
MOVL C01729 V=800.0 PL=0
MOVL C01730 V=800.0 PL=0
MOVL C01731 V=800.0 PL=0
MOVL C01732 V=800.0 PL=0
MOVL C01733 V=800.0 PL=0
MOVL C01734 V=800.0 PL=0
MOVL C01735 V=800.0 PL=0
MOVL C01736 V=800.0 PL=0
MOVL C01737 V=800.0 PL=0
MOVL C01738 V=800.0 PL=0
MOVL C01739 V=800.0 PL=0
MOVL C01740 V=800.0 PL=0
MOVL C01741 V=800.0 PL=0
MOVL C01742 V=800.0 PL=0
MOVL C01743 V=800.0 PL=0
MOVL C01744 V=800.0 PL=0
MOVL C01745 V=800.0 PL=0
MOVL C01746 V=800.0 PL=0
MOVL C01747 V=800.0 PL=0
MOVL C01748 V=800.0 PL=0
MOVL C01749 V=800.0 PL=0
MOVL C01750 V=800.0 PL=0
MOVL C01751 V=800.0 PL=0
MOVL C01752 V=800.0 PL=0
MOVL C01753 V=800.0 PL=0
MOVL C01754 V=800.0 PL=0
MOVL C01755 V=800.0 PL=0
MOVL C01756 V=800.0 PL=0
MOVL C01757 V=800.0 PL=0
MOVL C01758 V=800.0 PL=0
MOVL C01759 V=800.0 PL=0
MOVL C01760 V=800.0 PL=0
MOVL C01761 V=800.0 PL=0
MOVL C01762 V=800.0 PL=0
MOVL C01763 V=800.0 PL=0
MOVL C01764 V=800.0 PL=0
MOVL C01765 V=800.0 PL=0
MOVL C01766 V=800.0 PL=0
MOVL C01767 V=800.0 PL=0
MOVL C01768 V=800.0 PL=0
MOVL C01769 V=800.0 PL=0
MOVL C01770 V=800.0 PL=0
MOVL C01771 V=800.0 PL=0
MOVL C01772 V=800.0 PL=0
MOVL C01773 V=800.0 PL=0
MOVL C01774 V=800.0 PL=0
MOVL C01775 V=800.0 PL=0
MOVL C01776 V=800.0 PL=0
MOVL C01777 V=800.0 PL=0
MOVL C01778 V=800.0 PL=0
MOVL C01779 V=800.0 PL=0
MOVL C01780 V=800.0 PL=0
MOVL C01781 V=800.0 PL=0
MOVL C01782 V=800.0 PL=0
MOVL C01783 V=800.0 PL=0
MOVL C01784 V=800.0 PL=0
MOVL C01785 V=800.0 PL=0
MOVL C01786 V=800.0 PL=0
MOVL C01787 V=800.0 PL=0
MOVL C01788 V=800.0 PL=0
MOVL C01789 V=800.0 PL=0
MOVL C01790 V=800.0 PL=0
MOVL C01791 V=800.0 PL=0
MOVL C01792 V=800.0 PL=0
MOVL C01793 V=800.0 PL=0
MOVL C01794 V=800.0 PL=0
MOVL C01795 V=800.0 PL=0
MOVL C01796 V=800.0 PL=0
MOVL C01797 V=800.0 PL=0
MOVL C01798 V=800.0 PL=0
MOVL C01799 V=800.0 PL=0
MOVL C01800 V=800.0 PL=0
MOVL C01801 V=800.0 PL=0
MOVL C01802 V=800.0 PL=0
MOVL C01803 V=800.0 PL=0
MOVL C01804 V=800.0 PL=0
MOVL C01805 V=800.0 PL=0
MOVL C01806 V=800.0 PL=0
MOVL C01807 V=800.0 PL=0
MOVL C01808 V=800.0 PL=0
MOVL C01809 V=800.0 PL=0
MOVL C01810 V=800.0 PL=0
MOVL C01811 V=800.0 PL=0
MOVL C01812 V=800.0 PL=0
MOVL C01813 V=800.0 PL=0
MOVL C01814 V=800.0 PL=0
MOVL C01815 V=800.0 PL=0
MOVL C01816 V=800.0 PL=0
MOVL C01817 V=800.0 PL=0
MOVL C01818 V=800.0 PL=0
MOVL C01819 V=800.0 PL=0
MOVL C01820 V=800.0 PL=0
MOVL C01821 V=800.0 PL=0
MOVL C01822 V=800.0 PL=0
MOVL C01823 V=800.0 PL=0
MOVL C01824 V=800.0 PL=0
MOVL C01825 V=800.0 PL=0
MOVL C01826 V=800.0 PL=0
MOVL C01827 V=800.0 PL=0
MOVL C01828 V=800.0 PL=0
MOVL C01829 V=800.0 PL=0
MOVL C01830 V=800.0 PL=0
MOVL C01831 V=800.0 PL=0
MOVL C01832 V=800.0 PL=0
MOVL C01833 V=800.0 PL=0
MOVL C01834 V=800.0 PL=0
MOVL C01835 V=800.0 PL=0
MOVL C01836 V=800.0 PL=0
MOVL C01837 V=800.0 PL=0
MOVL C01838 V=800.0 PL=0
MOVL C01839 V=800.0 PL=0
MOVL C01840 V=800.0 PL=0
MOVL C01841 V=800.0 PL=0
MOVL C01842 V=800.0 PL=0
MOVL C01843 V=800.0 PL=0
MOVL C01844 V=800.0 PL=0
MOVL C01845 V=800.0 PL=0
MOVL C01846 V=800.0 PL=0
MOVL C01847 V=800.0 PL=0
MOVL C01848 V=800.0 PL=0
MOVL C01849 V=800.0 PL=0
MOVL C01850 V=800.0 PL=0
MOVL C01851 V=800.0 PL=0
MOVL C01852 V=800.0 PL=0
MOVL C01853 V=800.0 PL=0
MOVL C01854 V=800.0 PL=0
MOVL C01855 V=800.0 PL=0
MOVL C01856 V=800.0 PL=0
MOVL C01857 V=800.0 PL=0
MOVL C01858 V=800.0 PL=0
MOVL C01859 V=800.0 PL=0
MOVL C01860 V=800.0 PL=0
MOVL C01861 V=800.0 PL=0
MOVL C01862 V=800.0 PL=0
MOVL C01863 V=800.0 PL=0
MOVL C01864 V=800.0 PL=0
MOVL C01865 V=800.0 PL=0
MOVL C01866 V=800.0 PL=0
MOVL C01867 V=800.0 PL=0
MOVL C01868 V=800.0 PL=0
MOVL C01869 V=800.0 PL=0
MOVL C01870 V=800.0 PL=0
MOVL C01871 V=800.0 PL=0
MOVL C01872 V=800.0 PL=0
MOVL C01873 V=800.0 PL=0
MOVL C01874 V=800.0 PL=0
MOVL C01875 V=800.0 PL=0
MOVL C01876 V=800.0 PL=0
MOVL C01877 V=800.0 PL=0
MOVL C01878 V=800.0 PL=0
MOVL C01879 V=800.0 PL=0
MOVL C01880 V=800.0 PL=0
MOVL C01881 V=800.0 PL=0
MOVL C01882 V=800.0 PL=0
MOVL C01883 V=800.0 PL=0
MOVL C01884 V=800.0 PL=0
MOVL C01885 V=800.0 PL=0
MOVL C01886 V=800.0 PL=0
MOVL C01887 V=800.0 PL=0
MOVL C01888 V=800.0 PL=0
MOVL C01889 V=800.0 PL=0
MOVL C01890 V=800.0 PL=0
MOVL C01891 V=800.0 PL=0
MOVL C01892 V=800.0 PL=0
MOVL C01893 V=800.0 PL=0
MOVL C01894 V=800.0 PL=0
MOVL C01895 V=800.0 PL=0
MOVL C01896 V=800.0 PL=0
MOVL C01897 V=800.0 PL=0
MOVL C01898 V=800.0 PL=0
MOVL C01899 V=800.0 PL=0
MOVL C01900 V=800.0 PL=0
MOVL C01901 V=800.0 PL=0
MOVL C01902 V=800.0 PL=0
MOVL C01903 V=800.0 PL=0
MOVL C01904 V=800.0 PL=0
MOVL C01905 V=800.0 PL=0
MOVL C01906 V=800.0 PL=0
MOVL C01907 V=800.0 PL=0
MOVL C01908 V=800.0 PL=0
MOVL C01909 V=800.0 PL=0
MOVL C01910 V=800.0 PL=0
MOVL C01911 V=800.0 PL=0
MOVL C01912 V=800.0 PL=0
MOVL C01913 V=800.0 PL=0
MOVL C01914 V=800.0 PL=0
MOVL C01915 V=800.0 PL=0
MOVL C01916 V=800.0 PL=0
MOVL C01917 V=800.0 PL=0
MOVL C01918 V=800.0 PL=0
MOVL C01919 V=800.0 PL=0
MOVL C01920 V=800.0 PL=0
MOVL C01921 V=800.0 PL=0
MOVL C01922 V=800.0 PL=0
MOVL C01923 V=800.0 PL=0
MOVL C01924 V=800.0 PL=0
MOVL C01925 V=800.0 PL=0
MOVL C01926 V=800.0 PL=0
MOVL C01927 V=800.0 PL=0
MOVL C01928 V=800.0 PL=0
MOVL C01929 V=800.0 PL=0
MOVL C01930 V=800.0 PL=0
MOVL C01931 V=800.0 PL=0
MOVL C01932 V=800.0 PL=0
MOVL C01933 V=800.0 PL=0
MOVL C01934 V=800.0 PL=0
MOVL C01935 V=800.0 PL=0
MOVL C01936 V=800.0 PL=0
MOVL C01937 V=800.0 PL=0
MOVL C01938 V=800.0 PL=0
MOVL C01939 V=800.0 PL=0
MOVL C01940 V=800.0 PL=0
MOVL C01941 V=800.0 PL=0
MOVL C01942 V=800.0 PL=0
MOVL C01943 V=800.0 PL=0
MOVL C01944 V=800.0 PL=0
MOVL C01945 V=800.0 PL=0
MOVL C01946 V=800.0 PL=0
MOVL C01947 V=800.0 PL=0
MOVL C01948 V=800.0 PL=0
MOVL C01949 V=800.0 PL=0
MOVL C01950 V=800.0 PL=0
MOVL C01951 V=800.0 PL=0
MOVL C01952 V=800.0 PL=0
MOVL C01953 V=800.0 PL=0
MOVL C01954 V=800.0 PL=0
MOVL C01955 V=800.0 PL=0
MOVL C01956 V=800.0 PL=0
MOVL C01957 V=800.0 PL=0
MOVL C01958 V=800.0 PL=0
MOVL C01959 V=800.0 PL=0
MOVL C01960 V=800.0 PL=0
MOVL C01961 V=800.0 PL=0
MOVL C01962 V=800.0 PL=0
MOVL C01963 V=800.0 PL=0
MOVL C01964 V=800.0 PL=0
MOVL C01965 V=800.0 PL=0
MOVL C01966 V=800.0 PL=0
MOVL C01967 V=800.0 PL=0
MOVL C01968 V=800.0 PL=0
MOVL C01969 V=800.0 PL=0
MOVL C01970 V=800.0 PL=0
MOVL C01971 V=800.0 PL=0
MOVL C01972 V=800.0 PL=0
MOVL C01973 V=800.0 PL=0
MOVL C01974 V=800.0 PL=0
MOVL C01975 V=800.0 PL=0
MOVL C01976 V=800.0 PL=0
MOVL C01977 V=800.0 PL=0
MOVL C01978 V=800.0 PL=0
MOVL C01979 V=800.0 PL=0
MOVL C01980 V=800.0 PL=0
MOVL C01981 V=800.0 PL=0
MOVL C01982 V=800.0 PL=0
MOVL C01983 V=800.0 PL=0
MOVL C01984 V=800.0 PL=0
MOVL C01985 V=800.0 PL=0
MOVL C01986 V=800.0 PL=0
MOVL C01987 V=800.0 PL=0
MOVL C01988 V=800.0 PL=0
MOVL C01989 V=800.0 PL=0
MOVL C01990 V=800.0 PL=0
MOVL C01991 V=800.0 PL=0
MOVL C01992 V=800.0 PL=0
MOVL C01993 V=800.0 PL=0
MOVL C01994 V=800.0 PL=0
MOVL C01995 V=800.0 PL=0
